KUKA KRL program: MyProgram_283().src

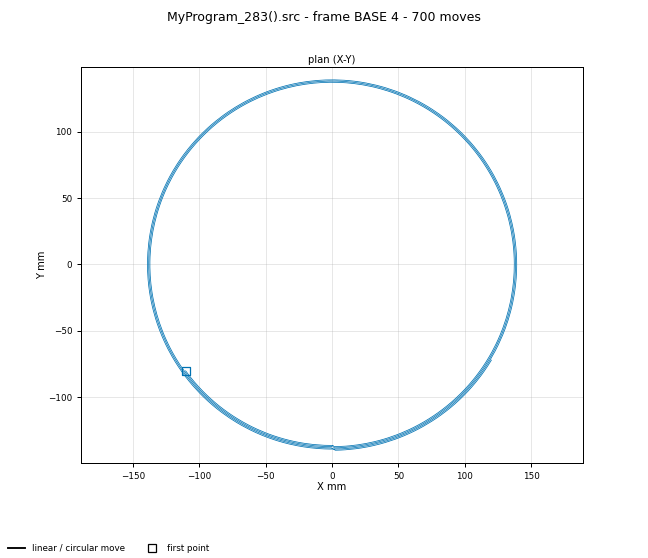
[picture p0: tool path of MyProgram_283().src in frame BASE 4, 700 of 700 moves have a stored position in this frame; points joined in program order, loops and branches not executed]
&ACCESS RVP
&REL 1
&PARAM TEMPLATE = C:\KRC\Roboter\Template\vorgabe
&PARAM EDITMASK = *
DEF MyProgram_283()
; ---- Setting reference (Base) ----
$BASE = BASE_DATA[4]

; --------------------------
; ---- Setting tool (TCP) ----
$TOOL = TOOL_DATA[3]
; --------------------------

$VEL.CP = VEL_APROX_PRINT
Startdeposition()
$VEL.CP = VEL_PRINT
LIN {X -110.2692,Y -80.0959,Z 174,A -140.9321,B 7.819,C 0.3265,E1 7.6978,E2 232.605} C_DIS
LIN {X -108.3483,Y -82.6759,Z 174,A -140.0536,B 7.8185,C 0.3365,E1 7.6992,E2 231.7869} C_DIS
LIN {X -106.4293,Y -85.1325,Z 174,A -138.4411,B 7.8186,C 0.3349,E1 7.7021,E2 230.1369} C_DIS
LIN {X -103.6871,Y -88.4515,Z 174,A -136.5544,B 7.8185,C 0.3377,E1 7.7055,E2 228.2411} C_DIS
LIN {X -100.4815,Y -92.0768,Z 174,A -134.4674,B 7.8184,C 0.3411,E1 7.7094,E2 226.1481} C_DIS
LIN {X -97.217,Y -95.517,Z 174,A -132.493,B 7.8182,C 0.3454,E1 7.7132,E2 224.1768} C_DIS
LIN {X -94.0859,Y -98.6027,Z 174,A -130.65,B 7.818,C 0.349,E1 7.7169,E2 222.335} C_DIS
LIN {X -91.5206,Y -100.9882,Z 174,A -129.1738,B 7.8179,C 0.3517,E1 7.7199,E2 220.8588} C_DIS
LIN {X -88.1965,Y -103.9039,Z 174,A -127.2223,B 7.8178,C 0.3537,E1 7.7241,E2 218.8959} C_DIS
LIN {X -85.404,Y -106.2113,Z 174,A -125.7546,B 7.8176,C 0.3571,E1 7.7273,E2 217.4355} C_DIS
LIN {X -81.9305,Y -108.9131,Z 174,A -123.8794,B 7.8176,C 0.3598,E1 7.7314,E2 215.5574} C_DIS
LIN {X -78.2052,Y -111.6189,Z 174,A -121.9045,B 7.8174,C 0.3623,E1 7.7359,E2 213.5778} C_DIS
LIN {X -74.5757,Y -114.0758,Z 174,A -119.9983,B 7.8174,C 0.3641,E1 7.7404,E2 211.6637} C_DIS
LIN {X -70.8017,Y -116.4554,Z 174,A -118.139,B 7.8172,C 0.367,E1 7.7448,E2 209.8066} C_DIS
LIN {X -67.0685,Y -118.6447,Z 174,A -116.2625,B 7.8172,C 0.3685,E1 7.7494,E2 207.9229} C_DIS
LIN {X -63.0831,Y -120.8085,Z 174,A -114.4681,B 7.8169,C 0.3727,E1 7.7537,E2 206.1427} C_DIS
LIN {X -59.9153,Y -122.4109,Z 174,A -112.95,B 7.8169,C 0.374,E1 7.7575,E2 204.6212} C_DIS
LIN {X -56.3626,Y -124.0885,Z 174,A -110.873,B 7.8171,C 0.369,E1 7.763,E2 202.4898} C_DIS
LIN {X -52.8036,Y -125.6422,Z 174,A -109.8689,B 7.8165,C 0.3809,E1 7.7653,E2 201.5659} C_DIS
LIN {X -50.2131,Y -126.7017,Z 174,A -108.4961,B 7.8166,C 0.3788,E1 7.769,E2 200.1681} C_DIS
LIN {X -47.4613,Y -127.7563,Z 174,A -107.243,B 7.8166,C 0.3797,E1 7.7722,E2 198.9129} C_DIS
LIN {X -43.8105,Y -129.0558,Z 174,A -105.3205,B 7.8167,C 0.3762,E1 7.7774,E2 196.9527} C_DIS
LIN {X -39.5544,Y -130.4212,Z 174,A -103.6952,B 7.8165,C 0.3818,E1 7.7817,E2 195.3594} C_DIS
LIN {X -36.2087,Y -131.39,Z 174,A -102.1521,B 7.8165,C 0.3815,E1 7.7858,E2 193.806} C_DIS
LIN {X -31.9644,Y -132.4856,Z 174,A -100.4334,B 7.8163,C 0.3847,E1 7.7905,E2 192.1027} C_DIS
LIN {X -28.5945,Y -133.2537,Z 174,A -98.9383,B 7.8163,C 0.3847,E1 7.7945,E2 190.6019} C_DIS
LIN {X -24.9403,Y -133.9873,Z 174,A -97.2215,B 7.8164,C 0.3828,E1 7.7993,E2 188.8655} C_DIS
LIN {X -20.6436,Y -134.7148,Z 174,A -95.52,B 7.8163,C 0.3857,E1 7.804,E2 187.18} C_DIS
LIN {X -13.919,Y -135.576,Z 174,A -92.555,B 7.8163,C 0.3844,E1 7.8122,E2 184.1995} C_DIS
LIN {X -5.8674,Y -136.1621,Z 174,A -88.2649,B 7.8171,C 0.3688,E1 7.8245,E2 179.7921} C_DIS
LIN {X 0.9737,Y -136.2785,Z 174,A -87.9401,B 7.8149,C 0.413,E1 7.8247,E2 179.7914} C_DIS
Enddeposition()
LIN {X 0.9737,Y -136.2785,Z 174,A -87.9404,B 7.8149,C 0.413,E1 7.8246,E2 179.7917} C_DIS
Startdeposition()
$VEL.CP = VEL_PRINT
LIN {X -0.4455,Y -137.1941,Z 174,A -87.6174,B 7.7989,C 0.4021,E1 7.8091,E2 179.393} C_DIS
LIN {X -3.8273,Y -137.1411,Z 174,A -88.9609,B 7.7989,C 0.401,E1 7.8053,E2 180.7283} C_DIS
LIN {X -6.8725,Y -137.0222,Z 174,A -90.2421,B 7.7989,C 0.4011,E1 7.8017,E2 182.0112} C_DIS
LIN {X -9.9728,Y -136.8314,Z 174,A -91.5485,B 7.7989,C 0.4011,E1 7.7981,E2 183.3192} C_DIS
LIN {X -13.3149,Y -136.5469,Z 174,A -93.0053,B 7.7989,C 0.4019,E1 7.794,E2 184.7837} C_DIS
LIN {X -17.0384,Y -136.1345,Z 174,A -94.5158,B 7.7989,C 0.4007,E1 7.7898,E2 186.288} C_DIS
LIN {X -19.6937,Y -135.7738,Z 174,A -95.6857,B 7.7989,C 0.4012,E1 7.7866,E2 187.4647} C_DIS
LIN {X -23.3734,Y -135.191,Z 174,A -97.2013,B 7.7989,C 0.4,E1 7.7824,E2 188.9758} C_DIS
LIN {X -25.9226,Y -134.723,Z 174,A -98.3187,B 7.7989,C 0.4001,E1 7.7793,E2 190.0978} C_DIS
LIN {X -29.7515,Y -133.9319,Z 174,A -99.9292,B 7.799,C 0.399,E1 7.775,E2 191.706} C_DIS
LIN {X -32.9498,Y -133.1812,Z 174,A -101.3082,B 7.799,C 0.3983,E1 7.7712,E2 193.0863} C_DIS
LIN {X -35.6372,Y -132.4851,Z 174,A -102.4768,B 7.799,C 0.3978,E1 7.768,E2 194.2562} C_DIS
LIN {X -39.3506,Y -131.4323,Z 174,A -104.0952,B 7.7991,C 0.3968,E1 7.7637,E2 195.8759} C_DIS
LIN {X -42.547,Y -130.4326,Z 174,A -105.5028,B 7.7991,C 0.3958,E1 7.76,E2 197.2848} C_DIS
LIN {X -45.2788,Y -129.5074,Z 174,A -106.7111,B 7.7992,C 0.3949,E1 7.7568,E2 198.4938} C_DIS
LIN {X -48.9163,Y -128.18,Z 174,A -108.344,B 7.7993,C 0.3937,E1 7.7525,E2 200.129} C_DIS
LIN {X -52.0827,Y -126.9264,Z 174,A -109.7771,B 7.7993,C 0.3925,E1 7.7488,E2 201.5636} C_DIS
LIN {X -55.2327,Y -125.5877,Z 174,A -111.2177,B 7.7994,C 0.3912,E1 7.7451,E2 203.0058} C_DIS
LIN {X -57.9714,Y -124.345,Z 174,A -112.4934,B 7.7994,C 0.3901,E1 7.7418,E2 204.284} C_DIS
LIN {X -61.4699,Y -122.6555,Z 174,A -114.1207,B 7.7996,C 0.3883,E1 7.7377,E2 205.912} C_DIS
LIN {X -64.5504,Y -121.0626,Z 174,A -115.5293,B 7.7996,C 0.3859,E1 7.7343,E2 207.3156} C_DIS
LIN {X -67.5416,Y -119.4194,Z 174,A -117.1085,B 7.7996,C 0.3865,E1 7.7304,E2 208.9142} C_DIS
LIN {X -71.3674,Y -117.1734,Z 174,A -118.9919,B 7.7998,C 0.3844,E1 7.7258,E2 210.8014} C_DIS
LIN {X -75.0753,Y -114.8329,Z 174,A -120.8424,B 7.7998,C 0.382,E1 7.7215,E2 212.6542} C_DIS
LIN {X -78.7185,Y -112.3668,Z 174,A -122.6965,B 7.8,C 0.3794,E1 7.7172,E2 214.5103} C_DIS
LIN {X -82.2906,Y -109.7778,Z 174,A -124.5598,B 7.8001,C 0.3768,E1 7.713,E2 216.3759} C_DIS
LIN {X -85.7856,Y -107.0689,Z 174,A -126.4313,B 7.8003,C 0.374,E1 7.7089,E2 218.2502} C_DIS
LIN {X -89.1974,Y -104.2437,Z 174,A -128.3004,B 7.8004,C 0.371,E1 7.7049,E2 220.1213} C_DIS
LIN {X -92.5203,Y -101.306,Z 174,A -130.1674,B 7.8006,C 0.3678,E1 7.701,E2 221.9898} C_DIS
LIN {X -95.7488,Y -98.2602,Z 174,A -132.0532,B 7.8007,C 0.3647,E1 7.6972,E2 223.8792} C_DIS
LIN {X -98.8778,Y -95.1109,Z 174,A -133.9317,B 7.8009,C 0.3614,E1 7.6936,E2 225.7601} C_DIS
LIN {X -101.9023,Y -91.8631,Z 174,A -135.8135,B 7.801,C 0.358,E1 7.69,E2 227.6449} C_DIS
LIN {X -104.8178,Y -88.5219,Z 174,A -137.691,B 7.8012,C 0.3545,E1 7.6866,E2 229.5249} C_DIS
LIN {X -107.6201,Y -85.093,Z 174,A -139.5665,B 7.8013,C 0.3508,E1 7.6833,E2 231.403} C_DIS
LIN {X -110.3053,Y -81.5822,Z 174,A -141.4389,B 7.8015,C 0.3471,E1 7.6801,E2 233.278} C_DIS
LIN {X -112.87,Y -77.9954,Z 174,A -143.3042,B 7.8017,C 0.3432,E1 7.6771,E2 235.1454} C_DIS
LIN {X -115.3112,Y -74.3387,Z 174,A -145.1385,B 7.8019,C 0.3388,E1 7.6743,E2 236.9785} C_DIS
LIN {X -117.6262,Y -70.6186,Z 174,A -147.0255,B 7.802,C 0.3352,E1 7.6716,E2 238.8718} C_DIS
LIN {X -119.8129,Y -66.8414,Z 174,A -148.8797,B 7.8022,C 0.3312,E1 7.669,E2 240.729} C_DIS
LIN {X -121.8696,Y -63.0137,Z 174,A -150.6229,B 7.8024,C 0.3256,E1 7.6668,E2 242.4622} C_DIS
LIN {X -123.252,Y -60.2605,Z 174,A -151.9559,B 7.8025,C 0.323,E1 7.6651,E2 243.8002} C_DIS
LIN {X -124.8864,Y -56.8005,Z 174,A -153.5542,B 7.8027,C 0.3189,E1 7.6632,E2 245.3976} C_DIS
LIN {X -126.2078,Y -53.7984,Z 174,A -154.9308,B 7.8028,C 0.3154,E1 7.6617,E2 246.7743} C_DIS
LIN {X -127.5638,Y -50.5013,Z 174,A -156.4598,B 7.803,C 0.3121,E1 7.6601,E2 248.3074} C_DIS
LIN {X -128.7749,Y -47.3279,Z 174,A -157.9017,B 7.8031,C 0.3086,E1 7.6587,E2 249.7512} C_DIS
LIN {X -129.8649,Y -44.2476,Z 174,A -159.2776,B 7.8032,C 0.3051,E1 7.6574,E2 251.1276} C_DIS
LIN {X -130.9429,Y -40.9494,Z 174,A -160.7629,B 7.8034,C 0.3016,E1 7.6561,E2 252.6164} C_DIS
LIN {X -131.9007,Y -37.7508,Z 174,A -162.1808,B 7.8035,C 0.2981,E1 7.655,E2 254.0363} C_DIS
LIN {X -132.775,Y -34.55,Z 174,A -163.5899,B 7.8036,C 0.2946,E1 7.654,E2 255.4473} C_DIS
LIN {X -133.5558,Y -31.3956,Z 174,A -164.9673,B 7.8038,C 0.2911,E1 7.6531,E2 256.8263} C_DIS
LIN {X -134.2131,Y -28.4489,Z 174,A -166.2332,B 7.8039,C 0.2877,E1 7.6524,E2 258.0917} C_DIS
LIN {X -134.9062,Y -24.9647,Z 174,A -167.9218,B 7.8039,C 0.2863,E1 7.6515,E2 259.8047} C_DIS
LIN {X -135.5635,Y -21.0908,Z 174,A -169.4474,B 7.8042,C 0.2801,E1 7.6508,E2 261.3146} C_DIS
LIN {X -136.0332,Y -17.8113,Z 174,A -170.838,B 7.8043,C 0.2762,E1 7.6502,E2 262.705} C_DIS
LIN {X -136.4086,Y -14.6623,Z 174,A -172.1793,B 7.8044,C 0.2727,E1 7.6498,E2 264.0473} C_DIS
LIN {X -136.7046,Y -11.5825,Z 174,A -173.5097,B 7.8045,C 0.2695,E1 7.6495,E2 265.3814} C_DIS
LIN {X -136.9358,Y -8.4199,Z 174,A -174.8471,B 7.8047,C 0.2659,E1 7.6492,E2 266.7192} C_DIS
LIN {X -137.0908,Y -5.331,Z 174,A -176.155,B 7.8047,C 0.2624,E1 7.6491,E2 268.0281} C_DIS
LIN {X -137.1758,Y -2.2664,Z 174,A -177.5113,B 7.8049,C 0.2598,E1 7.649,E2 269.3927} C_DIS
LIN {X -137.1758,Y 2.2664,Z 174,A -179.4228,B 7.805,C 0.2546,E1 7.649,E2 271.3049} C_DIS
LIN {X -137.0733,Y 5.7817,Z 174,A 179.0821,B 7.8052,C 0.2507,E1 7.6492,E2 272.8019} C_DIS
LIN {X -136.8871,Y 9.2111,Z 174,A 177.6403,B 7.8052,C 0.2467,E1 7.6494,E2 274.2435} C_DIS
LIN {X -136.6416,Y 12.3277,Z 174,A 176.3073,B 7.8054,C 0.2433,E1 7.6497,E2 275.5787} C_DIS
LIN {X -136.3398,Y 15.3018,Z 174,A 175.0369,B 7.8055,C 0.24,E1 7.6501,E2 276.8506} C_DIS
LIN {X -135.9783,Y 18.2303,Z 174,A 173.7751,B 7.8055,C 0.2369,E1 7.6505,E2 278.1149} C_DIS
LIN {X -135.456,Y 21.7848,Z 174,A 172.2427,B 7.8057,C 0.233,E1 7.6512,E2 279.6498} C_DIS
LIN {X -134.9062,Y 24.9647,Z 174,A 170.8671,B 7.8058,C 0.2296,E1 7.6519,E2 281.0276} C_DIS
LIN {X -134.2768,Y 28.1541,Z 174,A 169.4815,B 7.8059,C 0.2261,E1 7.6526,E2 282.4155} C_DIS
LIN {X -133.5668,Y 31.3501,Z 174,A 168.0864,B 7.806,C 0.2227,E1 7.6535,E2 283.8127} C_DIS
LIN {X -132.775,Y 34.55,Z 174,A 166.6818,B 7.8061,C 0.2192,E1 7.6545,E2 285.2193} C_DIS
LIN {X -131.9007,Y 37.7508,Z 174,A 165.2679,B 7.8062,C 0.2157,E1 7.6555,E2 286.6354} C_DIS
LIN {X -131.118,Y 40.3774,Z 174,A 164.0773,B 7.8062,C 0.2131,E1 7.6565,E2 287.8305} C_DIS
LIN {X -129.9012,Y 44.1428,Z 174,A 162.4156,B 7.8064,C 0.2087,E1 7.658,E2 289.4918} C_DIS
LIN {X -128.7749,Y 47.3279,Z 174,A 160.977,B 7.8064,C 0.2053,E1 7.6593,E2 290.9324} C_DIS
LIN {X -127.5638,Y 50.5013,Z 174,A 159.5313,B 7.8066,C 0.2018,E1 7.6608,E2 292.3801} C_DIS
LIN {X -126.2676,Y 53.66,Z 174,A 158.0783,B 7.8066,C 0.1984,E1 7.6624,E2 293.835} C_DIS
LIN {X -124.8864,Y 56.8005,Z 174,A 156.6188,B 7.8068,C 0.195,E1 7.664,E2 295.2964} C_DIS
LIN {X -123.4203,Y 59.9195,Z 174,A 155.1528,B 7.8068,C 0.1916,E1 7.6658,E2 296.7643} C_DIS
LIN {X -121.8696,Y 63.0137,Z 174,A 153.6811,B 7.8069,C 0.1882,E1 7.6677,E2 298.2377} C_DIS
LIN {X -120.4387,Y 65.7058,Z 174,A 152.3208,B 7.8069,C 0.1862,E1 7.6695,E2 299.6074} C_DIS
LIN {X -118.2905,Y 69.4987,Z 174,A 150.4681,B 7.8071,C 0.182,E1 7.6721,E2 301.4623} C_DIS
LIN {X -116.0135,Y 73.2364,Z 174,A 148.6087,B 7.8071,C 0.178,E1 7.6748,E2 303.3238} C_DIS
LIN {X -113.6097,Y 76.9126,Z 174,A 146.7435,B 7.8072,C 0.174,E1 7.6777,E2 305.191} C_DIS
LIN {X -111.1522,Y 80.4234,Z 174,A 144.8998,B 7.8073,C 0.1705,E1 7.6807,E2 307.0395} C_DIS
LIN {X -108.4431,Y 84.0405,Z 174,A 143.0035,B 7.8074,C 0.1663,E1 7.6839,E2 308.9351} C_DIS
LIN {X -105.6641,Y 87.5089,Z 174,A 141.1225,B 7.8074,C 0.1624,E1 7.6872,E2 310.8174} C_DIS
LIN {X -102.7942,Y 90.8629,Z 174,A 139.2504,B 7.8076,C 0.1588,E1 7.6906,E2 312.6912} C_DIS
LIN {X -99.7895,Y 94.1529,Z 174,A 137.3641,B 7.8076,C 0.1552,E1 7.6942,E2 314.5788} C_DIS
LIN {X -96.7042,Y 97.3191,Z 174,A 135.4889,B 7.8077,C 0.1518,E1 7.6979,E2 316.4558} C_DIS
LIN {X -93.5053,Y 100.3966,Z 174,A 133.6105,B 7.8077,C 0.1485,E1 7.7017,E2 318.3355} C_DIS
LIN {X -90.1964,Y 103.3795,Z 174,A 131.7333,B 7.8078,C 0.1451,E1 7.7056,E2 320.213} C_DIS
LIN {X -86.8106,Y 106.2386,Z 174,A 129.8571,B 7.8078,C 0.1421,E1 7.7097,E2 322.0907} C_DIS
LIN {X -83.3398,Y 108.9825,Z 174,A 127.9883,B 7.8079,C 0.1391,E1 7.7138,E2 323.9604} C_DIS
LIN {X -79.7901,Y 111.6076,Z 174,A 126.1244,B 7.8079,C 0.1362,E1 7.718,E2 325.8252} C_DIS
LIN {X -76.1826,Y 114.1005,Z 174,A 124.2709,B 7.808,C 0.1336,E1 7.7223,E2 327.6797} C_DIS
LIN {X -72.4936,Y 116.4792,Z 174,A 122.4202,B 7.808,C 0.131,E1 7.7266,E2 329.531} C_DIS
LIN {X -68.7443,Y 118.7305,Z 174,A 120.5776,B 7.8081,C 0.1285,E1 7.7311,E2 331.3741} C_DIS
LIN {X -65.1753,Y 120.7269,Z 174,A 118.7981,B 7.8081,C 0.1272,E1 7.7354,E2 333.1609} C_DIS
LIN {X -61.6024,Y 122.588,Z 174,A 117.2225,B 7.8082,C 0.1234,E1 7.7393,E2 334.7222} C_DIS
LIN {X -58.3628,Y 124.164,Z 174,A 115.7112,B 7.8082,C 0.1216,E1 7.7431,E2 336.2332} C_DIS
LIN {X -55.5354,Y 125.4523,Z 174,A 114.3848,B 7.8082,C 0.1205,E1 7.7465,E2 337.562} C_DIS
LIN {X -52.0827,Y 126.9264,Z 174,A 112.8269,B 7.8082,C 0.1186,E1 7.7505,E2 339.1176} C_DIS
LIN {X -49.2458,Y 128.0519,Z 174,A 111.5224,B 7.8082,C 0.1177,E1 7.7539,E2 340.4247} C_DIS
LIN {X -45.7366,Y 129.3487,Z 174,A 109.9741,B 7.8083,C 0.1159,E1 7.758,E2 341.9702} C_DIS
LIN {X -43.1013,Y 130.248,Z 174,A 108.7904,B 7.8083,C 0.1152,E1 7.7611,E2 343.1556} C_DIS
LIN {X -39.7978,Y 131.2954,Z 174,A 107.3456,B 7.8083,C 0.1139,E1 7.765,E2 344.5991} C_DIS
LIN {X -36.1505,Y 132.3482,Z 174,A 105.7605,B 7.8083,C 0.1126,E1 7.7692,E2 346.1832} C_DIS
LIN {X -33.2373,Y 133.1082,Z 174,A 104.5097,B 7.8083,C 0.1116,E1 7.7726,E2 347.4323} C_DIS
LIN {X -29.7515,Y 133.9319,Z 174,A 102.9992,B 7.8083,C 0.1109,E1 7.7767,E2 348.9437} C_DIS
LIN {X -26.5584,Y 134.6015,Z 174,A 101.6336,B 7.8083,C 0.1102,E1 7.7805,E2 350.3089} C_DIS
LIN {X -23.3734,Y 135.191,Z 174,A 100.2786,B 7.8084,C 0.1095,E1 7.7842,E2 351.6634} C_DIS
LIN {X -20.5736,Y 135.6436,Z 174,A 99.1141,B 7.8084,C 0.1086,E1 7.7874,E2 352.8246} C_DIS
LIN {X -17.0384,Y 136.1345,Z 174,A 97.601,B 7.8084,C 0.1084,E1 7.7916,E2 354.3398} C_DIS
LIN {X -13.8935,Y 136.4913,Z 174,A 96.2787,B 7.8084,C 0.108,E1 7.7952,E2 355.6614} C_DIS
LIN {X -10.7669,Y 136.7735,Z 174,A 94.9682,B 7.8084,C 0.1077,E1 7.7989,E2 356.9712} C_DIS
LIN {X -7.6609,Y 136.9826,Z 174,A 93.6688,B 7.8084,C 0.1074,E1 7.8025,E2 358.2698} C_DIS
LIN {X -4.6128,Y 137.1189,Z 174,A 92.3958,B 7.8084,C 0.1073,E1 7.8061,E2 359.542} C_DIS
LIN {X -1.5193,Y 137.1882,Z 174,A 91.1061,B 7.8084,C 0.1072,E1 7.8097,E2 360.8308} C_DIS
LIN {X 1.5193,Y 137.1882,Z 174,A 89.8358,B 7.8084,C 0.1072,E1 7.8132,E2 362.1007} C_DIS
LIN {X 4.5776,Y 137.1202,Z 174,A 88.5564,B 7.8084,C 0.1073,E1 7.8168,E2 363.3799} C_DIS
LIN {X 7.6609,Y 136.9826,Z 174,A 87.2662,B 7.8084,C 0.1075,E1 7.8204,E2 364.6696} C_DIS
LIN {X 10.7669,Y 136.7735,Z 174,A 85.9654,B 7.8084,C 0.1078,E1 7.824,E2 365.9701} C_DIS
LIN {X 13.8935,Y 136.4913,Z 174,A 84.6542,B 7.8084,C 0.1082,E1 7.8276,E2 367.2808} C_DIS
LIN {X 16.4844,Y 136.2006,Z 174,A 83.5114,B 7.8084,C 0.1094,E1 7.8308,E2 368.4298} C_DIS
LIN {X 20.1992,Y 135.7015,Z 174,A 82.0017,B 7.8084,C 0.1091,E1 7.835,E2 369.9322} C_DIS
LIN {X 23.02,Y 135.2499,Z 174,A 80.8055,B 7.8084,C 0.1097,E1 7.8383,E2 371.1284} C_DIS
LIN {X 26.5584,Y 134.6015,Z 174,A 79.3107,B 7.8084,C 0.1104,E1 7.8424,E2 372.6219} C_DIS
LIN {X 29.7515,Y 133.9319,Z 174,A 77.9513,B 7.8084,C 0.1112,E1 7.8461,E2 373.9806} C_DIS
LIN {X 32.4849,Y 133.2932,Z 174,A 76.7795,B 7.8084,C 0.1119,E1 7.8493,E2 375.1519} C_DIS
LIN {X 36.1505,Y 132.3482,Z 174,A 75.2069,B 7.8084,C 0.1129,E1 7.8535,E2 376.7233} C_DIS
LIN {X 39.3506,Y 131.4323,Z 174,A 73.8223,B 7.8084,C 0.114,E1 7.8572,E2 378.107} C_DIS
LIN {X 42.1496,Y 130.5595,Z 174,A 72.6051,B 7.8084,C 0.1149,E1 7.8605,E2 379.323} C_DIS
LIN {X 45.3005,Y 129.4999,Z 174,A 71.184,B 7.8084,C 0.1168,E1 7.8642,E2 380.7478} C_DIS
LIN {X 48.9163,Y 128.18,Z 174,A 69.6223,B 7.8083,C 0.1176,E1 7.8683,E2 382.3038} C_DIS
LIN {X 52.0827,Y 126.9264,Z 174,A 68.2082,B 7.8083,C 0.1189,E1 7.872,E2 383.7168} C_DIS
LIN {X 54.7796,Y 125.7835,Z 174,A 66.971,B 7.8083,C 0.1206,E1 7.8751,E2 384.9555} C_DIS
LIN {X 58.3628,Y 124.164,Z 174,A 65.3616,B 7.8083,C 0.1219,E1 7.8792,E2 386.561} C_DIS
LIN {X 61.4699,Y 122.6555,Z 174,A 63.9296,B 7.8082,C 0.1236,E1 7.8828,E2 387.9916} C_DIS
LIN {X 65.316,Y 120.6513,Z 174,A 62.0347,B 7.8082,C 0.1275,E1 7.8875,E2 389.8968} C_DIS
LIN {X 69.1142,Y 118.5164,Z 174,A 60.2332,B 7.8081,C 0.1298,E1 7.8919,E2 391.6961} C_DIS
LIN {X 72.8152,Y 116.279,Z 174,A 58.4343,B 7.8081,C 0.1324,E1 7.8961,E2 393.4943} C_DIS
LIN {X 76.5407,Y 113.8614,Z 174,A 56.6028,B 7.8081,C 0.1349,E1 7.9004,E2 395.3232} C_DIS
LIN {X 80.1165,Y 111.3742,Z 174,A 54.8001,B 7.808,C 0.1376,E1 7.9045,E2 397.1241} C_DIS
LIN {X 83.6439,Y 108.75,Z 174,A 52.981,B 7.808,C 0.1404,E1 7.9086,E2 398.9413} C_DIS
LIN {X 87.1606,Y 105.9525,Z 174,A 51.1526,B 7.8079,C 0.1429,E1 7.9125,E2 400.7642} C_DIS
LIN {X 90.5375,Y 103.0819,Z 174,A 49.3008,B 7.8079,C 0.1464,E1 7.9164,E2 402.6166} C_DIS
LIN {X 93.8233,Y 100.1004,Z 174,A 47.474,B 7.8077,C 0.1495,E1 7.9202,E2 404.4406} C_DIS
LIN {X 97.0127,Y 97.0127,Z 174,A 45.6408,B 7.8077,C 0.1528,E1 7.9238,E2 406.2718} C_DIS
LIN {X 100.1004,Y 93.8233,Z 174,A 43.8151,B 7.8077,C 0.1561,E1 7.9273,E2 408.0947} C_DIS
LIN {X 103.0484,Y 90.5753,Z 174,A 42.0001,B 7.8075,C 0.1597,E1 7.9307,E2 409.9081} C_DIS
LIN {X 105.9525,Y 87.1606,Z 174,A 40.1605,B 7.8075,C 0.1632,E1 7.934,E2 411.7444} C_DIS
LIN {X 108.7084,Y 83.6982,Z 174,A 38.3433,B 7.8075,C 0.1668,E1 7.9371,E2 413.5585} C_DIS
LIN {X 111.3458,Y 80.1562,Z 174,A 36.5276,B 7.8073,C 0.1705,E1 7.9401,E2 415.3716} C_DIS
LIN {X 113.8614,Y 76.5407,Z 174,A 34.7284,B 7.8073,C 0.174,E1 7.9429,E2 417.1667} C_DIS
LIN {X 116.2257,Y 72.9003,Z 174,A 32.9254,B 7.8071,C 0.1782,E1 7.9456,E2 418.9693} C_DIS
LIN {X 118.5164,Y 69.1142,Z 174,A 31.1171,B 7.8071,C 0.182,E1 7.9482,E2 420.7737} C_DIS
LIN {X 120.6905,Y 65.243,Z 174,A 29.2721,B 7.807,C 0.1865,E1 7.9507,E2 422.6184} C_DIS
LIN {X 122.6555,Y 61.4699,Z 174,A 27.6419,B 7.807,C 0.1881,E1 7.9528,E2 424.2315} C_DIS
LIN {X 124.06,Y 58.5804,Z 174,A 26.3164,B 7.8068,C 0.1913,E1 7.9544,E2 425.5558} C_DIS
LIN {X 125.5877,Y 55.2327,Z 174,A 24.8144,B 7.8068,C 0.1946,E1 7.9561,E2 427.0544} C_DIS
LIN {X 126.9264,Y 52.0827,Z 174,A 23.4107,B 7.8067,C 0.1979,E1 7.9576,E2 428.4558} C_DIS
LIN {X 128.18,Y 48.9163,Z 174,A 22.0147,B 7.8066,C 0.2012,E1 7.959,E2 429.8495} C_DIS
LIN {X 129.3071,Y 45.852,Z 174,A 20.6839,B 7.8066,C 0.2042,E1 7.9602,E2 431.177} C_DIS
LIN {X 130.291,Y 42.9722,Z 174,A 19.3951,B 7.8064,C 0.208,E1 7.9614,E2 432.4689} C_DIS
LIN {X 131.4323,Y 39.3506,Z 174,A 17.8735,B 7.8064,C 0.2111,E1 7.9626,E2 433.9837} C_DIS
LIN {X 132.2311,Y 36.5694,Z 174,A 16.7076,B 7.8063,C 0.2136,E1 7.9635,E2 435.145} C_DIS
LIN {X 133.0818,Y 33.3411,Z 174,A 15.2919,B 7.8061,C 0.2179,E1 7.9645,E2 436.5644} C_DIS
LIN {X 133.9319,Y 29.7515,Z 174,A 13.81,B 7.8061,C 0.221,E1 7.9654,E2 438.0403} C_DIS
LIN {X 134.5149,Y 26.9838,Z 174,A 12.6419,B 7.806,C 0.2241,E1 7.9661,E2 439.2076} C_DIS
LIN {X 135.1366,Y 23.6773,Z 174,A 11.2568,B 7.8059,C 0.2277,E1 7.9668,E2 440.5912} C_DIS
LIN {X 135.7015,Y 20.1992,Z 174,A 9.8324,B 7.8058,C 0.2309,E1 7.9674,E2 442.011} C_DIS
LIN {X 136.1345,Y 17.0384,Z 174,A 8.5267,B 7.8057,C 0.2342,E1 7.9679,E2 443.3145} C_DIS
LIN {X 136.4913,Y 13.8935,Z 174,A 7.2313,B 7.8056,C 0.2374,E1 7.9683,E2 444.6076} C_DIS
LIN {X 136.7233,Y 11.3606,Z 174,A 6.1315,B 7.8055,C 0.2412,E1 7.9685,E2 445.713} C_DIS
LIN {X 136.9826,Y 7.6609,Z 174,A 4.6731,B 7.8054,C 0.2439,E1 7.9688,E2 447.1614} C_DIS
LIN {X 137.1352,Y 4.0399,Z 174,A 3.1415,B 7.8052,C 0.2486,E1 7.9689,E2 448.6964} C_DIS
LIN {X 137.196,Y 0.3997,Z 174,A 1.6281,B 7.8052,C 0.2528,E1 7.9689,E2 450.2104} C_DIS
LIN {X 137.1628,Y -3.0452,Z 174,A 0.2856,B 7.805,C 0.2551,E1 7.9689,E2 451.5421} C_DIS
LIN {X 137.0602,Y -6.1163,Z 174,A -0.9764,B 7.805,C 0.2583,E1 7.9688,E2 452.8026} C_DIS
LIN {X 136.8871,Y -9.2111,Z 174,A -2.2496,B 7.8048,C 0.2616,E1 7.9686,E2 454.0743} C_DIS
LIN {X 136.6416,Y -12.3277,Z 174,A -3.5333,B 7.8048,C 0.2649,E1 7.9683,E2 455.3563} C_DIS
LIN {X 136.3336,Y -15.3591,Z 174,A -4.7733,B 7.8046,C 0.268,E1 7.9679,E2 456.5935} C_DIS
LIN {X 135.9276,Y -18.6169,Z 174,A -6.133,B 7.8045,C 0.2717,E1 7.9674,E2 457.9529} C_DIS
LIN {X 135.456,Y -21.7848,Z 174,A -7.448,B 7.8044,C 0.275,E1 7.9668,E2 459.2664} C_DIS
LIN {X 134.9062,Y -24.9647,Z 174,A -8.7732,B 7.8042,C 0.2784,E1 7.9662,E2 460.59} C_DIS
LIN {X 134.3758,Y -27.6674,Z 174,A -9.9471,B 7.8042,C 0.2822,E1 7.9655,E2 461.7679} C_DIS
LIN {X 133.5668,Y -31.3501,Z 174,A -11.4528,B 7.804,C 0.2852,E1 7.9646,E2 463.2664} C_DIS
LIN {X 132.8048,Y -34.4326,Z 174,A -12.7599,B 7.8039,C 0.2886,E1 7.9637,E2 464.5725} C_DIS
LIN {X 131.9007,Y -37.7508,Z 174,A -14.1696,B 7.8037,C 0.2921,E1 7.9627,E2 465.9802} C_DIS
LIN {X 130.9429,Y -40.9494,Z 174,A -15.541,B 7.8037,C 0.2955,E1 7.9616,E2 467.35} C_DIS
LIN {X 129.9012,Y -44.1428,Z 174,A -16.9205,B 7.8035,C 0.2989,E1 7.9603,E2 468.7279} C_DIS
LIN {X 128.7749,Y -47.3279,Z 174,A -18.3084,B 7.8034,C 0.3023,E1 7.959,E2 470.1144} C_DIS
LIN {X 127.6321,Y -50.3256,Z 174,A -19.6165,B 7.8032,C 0.3053,E1 7.9577,E2 471.4198} C_DIS
LIN {X 126.2676,Y -53.66,Z 174,A -21.1065,B 7.8031,C 0.3091,E1 7.9561,E2 472.9094} C_DIS
LIN {X 124.8864,Y -56.8005,Z 174,A -22.5161,B 7.803,C 0.3124,E1 7.9545,E2 474.3175} C_DIS
LIN {X 123.4203,Y -59.9195,Z 174,A -23.9324,B 7.8028,C 0.3158,E1 7.9528,E2 475.7324} C_DIS
LIN {X 121.8696,Y -63.0137,Z 174,A -25.3549,B 7.8027,C 0.3191,E1 7.951,E2 477.1533} C_DIS
LIN {X 120.4387,Y -65.7058,Z 174,A -26.6698,B 7.8025,C 0.3232,E1 7.9493,E2 478.4748} C_DIS
LIN {X 118.2905,Y -69.4987,Z 174,A -28.4621,B 7.8024,C 0.3273,E1 7.9468,E2 480.2653} C_DIS
LIN {X 116.0135,Y -73.2364,Z 174,A -30.262,B 7.8022,C 0.3313,E1 7.9441,E2 482.0635} C_DIS
LIN {X 113.6097,Y -76.9126,Z 174,A -32.0686,B 7.802,C 0.3353,E1 7.9413,E2 483.8684} C_DIS
LIN {X 111.0923,Y -80.506,Z 174,A -33.8771,B 7.8018,C 0.3392,E1 7.9384,E2 485.6757} C_DIS
LIN {X 108.4431,Y -84.0405,Z 174,A -35.6948,B 7.8017,C 0.343,E1 7.9353,E2 487.4918} C_DIS
LIN {X 105.6641,Y -87.5089,Z 174,A -37.5207,B 7.8015,C 0.3467,E1 7.9321,E2 489.3156} C_DIS
LIN {X 102.7942,Y -90.8629,Z 174,A -39.3416,B 7.8014,C 0.3504,E1 7.9288,E2 491.1354} C_DIS
LIN {X 99.7895,Y -94.1529,Z 174,A -41.1729,B 7.8012,C 0.3539,E1 7.9253,E2 492.9648} C_DIS
LIN {X 96.7515,Y -97.2722,Z 174,A -42.983,B 7.801,C 0.3576,E1 7.9218,E2 494.7756} C_DIS
LIN {X 93.5053,Y -100.3966,Z 174,A -44.8265,B 7.8009,C 0.3607,E1 7.918,E2 496.616} C_DIS
LIN {X 90.1964,Y -103.3795,Z 174,A -46.6592,B 7.8007,C 0.3639,E1 7.9142,E2 498.4469} C_DIS
LIN {X 86.911,Y -106.1565,Z 174,A -48.4587,B 7.8006,C 0.3674,E1 7.9103,E2 500.2484} C_DIS
LIN {X 83.3398,Y -108.9825,Z 174,A -50.3112,B 7.8005,C 0.37,E1 7.9063,E2 502.0964} C_DIS
LIN {X 79.7901,Y -111.6076,Z 174,A -52.133,B 7.8003,C 0.3729,E1 7.9021,E2 503.917} C_DIS
LIN {X 76.2021,Y -114.0875,Z 174,A -53.9411,B 7.8002,C 0.3757,E1 7.898,E2 505.7251} C_DIS
LIN {X 72.4936,Y -116.4792,Z 174,A -55.7587,B 7.8001,C 0.3783,E1 7.8937,E2 507.541} C_DIS
LIN {X 68.7443,Y -118.7305,Z 174,A -57.565,B 7.7999,C 0.3807,E1 7.8893,E2 509.3463} C_DIS
LIN {X 64.9253,Y -120.8612,Z 174,A -59.3579,B 7.7999,C 0.3828,E1 7.885,E2 511.1365} C_DIS
LIN {X 61.4699,Y -122.6555,Z 174,A -60.9165,B 7.7998,C 0.3839,E1 7.8811,E2 512.6879} C_DIS
LIN {X 58.3628,Y -124.164,Z 174,A -62.3451,B 7.7998,C 0.3856,E1 7.8775,E2 514.1158} C_DIS
LIN {X 55.2327,Y -125.5877,Z 174,A -63.7677,B 7.7996,C 0.3871,E1 7.8739,E2 515.5378} C_DIS
LIN {X 52.4956,Y -126.7539,Z 174,A -65.033,B 7.7996,C 0.3891,E1 7.8706,E2 516.8069} C_DIS
LIN {X 48.9163,Y -128.18,Z 174,A -66.5941,B 7.7995,C 0.3901,E1 7.8666,E2 518.3632} C_DIS
LIN {X 45.7366,Y -129.3487,Z 174,A -67.9974,B 7.7995,C 0.3914,E1 7.8629,E2 519.7661} C_DIS
LIN {X 42.547,Y -130.4326,Z 174,A -69.3929,B 7.7994,C 0.3926,E1 7.8592,E2 521.1612} C_DIS
LIN {X 39.5764,Y -131.3631,Z 174,A -70.6937,B 7.7993,C 0.3939,E1 7.8557,E2 522.4629} C_DIS
LIN {X 36.1505,Y -132.3482,Z 174,A -72.1614,B 7.7993,C 0.3948,E1 7.8518,E2 523.929} C_DIS
LIN {X 32.1666,Y -133.37,Z 174,A -73.8669,B 7.7992,C 0.396,E1 7.8471,E2 525.634} C_DIS
LIN {X 28.9694,Y -134.1008,Z 174,A -75.2342,B 7.7992,C 0.397,E1 7.8434,E2 527.0019} C_DIS
LIN {X 25.7781,Y -134.7507,Z 174,A -76.5797,B 7.7992,C 0.3976,E1 7.8397,E2 528.3465} C_DIS
LIN {X 22.5956,Y -135.3207,Z 174,A -77.9225,B 7.7991,C 0.3983,E1 7.836,E2 529.6891} C_DIS
LIN {X 19.4245,Y -135.8122,Z 174,A -79.2619,B 7.7991,C 0.399,E1 7.8323,E2 531.0292} C_DIS
LIN {X 16.2347,Y -136.2304,Z 174,A -80.5926,B 7.7991,C 0.3995,E1 7.8287,E2 532.359} C_DIS
LIN {X 13.1269,Y -136.5649,Z 174,A -81.8919,B 7.799,C 0.3999,E1 7.825,E2 533.6583} C_DIS
LIN {X 9.9728,Y -136.8314,Z 174,A -83.2417,B 7.799,C 0.4008,E1 7.8213,E2 535.0124} C_DIS
LIN {X 6.1163,Y -137.0602,Z 174,A -84.8167,B 7.799,C 0.4006,E1 7.8169,E2 536.5834} C_DIS
LIN {X 3.0452,Y -137.1628,Z 174,A -86.0956,B 7.799,C 0.4008,E1 7.8133,E2 537.8624} C_DIS
LIN {X 0.9766,Y -137.1895,Z 174,A -86.8725,B 7.799,C 0.3994,E1 7.8112,E2 538.6284} C_DIS
Enddeposition()
LIN {X 0.9766,Y -137.1895,Z 174,A -86.8725,B 7.799,C 0.3994,E1 7.8112,E2 538.6284} C_DIS
Startdeposition()
$VEL.CP = VEL_PRINT
LIN {X 1.6084,Y -138.094,Z 174,A -85.9601,B 7.782,C 0.3926,E1 7.7965,E2 537.6704} C_DIS
LIN {X 5.5097,Y -137.9917,Z 174,A -84.4095,B 7.782,C 0.3935,E1 7.8008,E2 536.1279} C_DIS
LIN {X 9.8394,Y -137.7507,Z 174,A -82.6213,B 7.782,C 0.3931,E1 7.8058,E2 534.3401} C_DIS
LIN {X 13.4506,Y -137.4451,Z 174,A -81.1698,B 7.782,C 0.3935,E1 7.8098,E2 532.8947} C_DIS
LIN {X 16.6463,Y -137.0948,Z 174,A -79.0849,B 7.7826,C 0.3792,E1 7.8159,E2 530.7105} C_DIS
LIN {X 22.351,Y -136.2812,Z 174,A -77.6149,B 7.7818,C 0.3947,E1 7.8196,E2 529.3597} C_DIS
LIN {X 26.3325,Y -135.5682,Z 174,A -75.8066,B 7.782,C 0.3912,E1 7.8246,E2 527.5335} C_DIS
LIN {X 29.4156,Y -134.9325,Z 174,A -74.4572,B 7.7821,C 0.3895,E1 7.8283,E2 526.1776} C_DIS
LIN {X 34.0037,Y -133.8496,Z 174,A -72.5109,B 7.7821,C 0.3881,E1 7.8336,E2 524.2312} C_DIS
LIN {X 37.0264,Y -133.0452,Z 174,A -71.2168,B 7.7822,C 0.3871,E1 7.8371,E2 522.9367} C_DIS
LIN {X 40.3618,Y -132.0714,Z 174,A -69.8055,B 7.7822,C 0.3863,E1 7.8408,E2 521.5284} C_DIS
LIN {X 45.7189,Y -130.3149,Z 174,A -67.4739,B 7.7824,C 0.384,E1 7.847,E2 519.1961} C_DIS
LIN {X 50.7038,Y -128.4581,Z 174,A -65.3045,B 7.7824,C 0.3822,E1 7.8527,E2 517.03} C_DIS
LIN {X 53.4133,Y -127.3537,Z 174,A -63.8756,B 7.7827,C 0.3767,E1 7.8564,E2 515.572} C_DIS
LIN {X 58.3037,Y -125.1907,Z 174,A -61.8635,B 7.7827,C 0.3777,E1 7.8615,E2 513.5852} C_DIS
LIN {X 61.9206,Y -123.4439,Z 174,A -60.2432,B 7.7827,C 0.3763,E1 7.8655,E2 511.9696} C_DIS
LIN {X 65.5374,Y -121.5621,Z 174,A -58.4935,B 7.7829,C 0.3728,E1 7.8699,E2 510.2109} C_DIS
LIN {X 69.2755,Y -119.4712,Z 174,A -56.4123,B 7.7833,C 0.3642,E1 7.875,E2 508.0884} C_DIS
LIN {X 72.5939,Y -117.4851,Z 174,A -55.0773,B 7.7833,C 0.3668,E1 7.8781,E2 506.7872} C_DIS
LIN {X 76.3802,Y -115.0593,Z 174,A -53.2717,B 7.7833,C 0.3649,E1 7.8823,E2 504.9878} C_DIS
LIN {X 80.6698,Y -112.0938,Z 174,A -50.14,B 7.7843,C 0.342,E1 7.8897,E2 501.727} C_DIS
LIN {X 86.7659,Y -107.4436,Z 174,A -48.4205,B 7.7833,C 0.3649,E1 7.8931,E2 500.1961} C_DIS
LIN {X 92.5399,Y -102.5131,Z 174,A -45.1507,B 7.7837,C 0.3564,E1 7.9001,E2 496.9081} C_DIS
LIN {X 96.8835,Y -98.4179,Z 174,A -42.5618,B 7.784,C 0.3491,E1 7.9053,E2 494.3024} C_DIS
LIN {X 102.454,Y -92.6051,Z 174,A -38.932,B 7.7846,C 0.3361,E1 7.9123,E2 490.6319} C_DIS
LIN {X 104.6651,Y -90.0981,Z 174,A -37.8424,B 7.7845,C 0.3389,E1 7.9143,E2 489.5797} C_DIS
LIN {X 107.2864,Y -86.9608,Z 174,A -35.7737,B 7.7849,C 0.3275,E1 7.918,E2 487.4609} C_DIS
LIN {X 109.7627,Y -83.813,Z 174,A -34.62,B 7.7847,C 0.3339,E1 7.9199,E2 486.3716} C_DIS
LIN {X 111.3156,Y -81.7391,Z 174,A -33.432,B 7.7849,C 0.329,E1 7.9219,E2 485.1679} C_DIS
LIN {X 113.8492,Y -78.1716,Z 174,A -31.6261,B 7.7851,C 0.3248,E1 7.9247,E2 483.3614} C_DIS
LIN {X 116.1827,Y -74.6598,Z 174,A -29.8936,B 7.7852,C 0.3209,E1 7.9274,E2 481.6294} C_DIS
LIN {X 118.6352,Y -70.6974,Z 174,A -28.0055,B 7.7854,C 0.3169,E1 7.9301,E2 479.7452} C_DIS
LIN {X 120.7887,Y -66.9517,Z 174,A -26.2425,B 7.7855,C 0.3129,E1 7.9325,E2 477.9843} C_DIS
LIN {X 123.1866,Y -62.4261,Z 174,A -24.1983,B 7.7857,C 0.309,E1 7.9352,E2 475.9484} C_DIS
LIN {X 126.4305,Y -55.5691,Z 174,A -21.1486,B 7.7859,C 0.3027,E1 7.9387,E2 472.9084} C_DIS
LIN {X 128.0379,Y -51.7514,Z 174,A -19.1525,B 7.7863,C 0.2924,E1 7.9409,E2 470.8745} C_DIS
LIN {X 129.264,Y -48.6083,Z 174,A -18.3195,B 7.786,C 0.3001,E1 7.9417,E2 470.1134} C_DIS
LIN {X 130.5829,Y -44.9458,Z 174,A -16.4899,B 7.7864,C 0.2913,E1 7.9434,E2 468.2545} C_DIS
LIN {X 131.732,Y -41.4604,Z 174,A -14.5054,B 7.7869,C 0.2776,E1 7.9451,E2 466.2087} C_DIS
LIN {X 132.9701,Y -37.2951,Z 174,A -13.1956,B 7.7867,C 0.2827,E1 7.9461,E2 464.961} C_DIS
LIN {X 134.032,Y -33.285,Z 174,A -11.5341,B 7.7868,C 0.2791,E1 7.9472,E2 463.3057} C_DIS
LIN {X 134.8398,Y -29.8447,Z 174,A -10.0633,B 7.787,C 0.2748,E1 7.9481,E2 461.8328} C_DIS
LIN {X 135.8403,Y -24.8945,Z 174,A -7.0678,B 7.7878,C 0.2503,E1 7.9497,E2 458.7185} C_DIS
LIN {X 136.932,Y -17.9345,Z 174,A -5.1962,B 7.7874,C 0.2636,E1 7.9504,E2 456.9805} C_DIS
LIN {X 137.7575,Y -9.7468,Z 174,A -1.098,B 7.7881,C 0.2397,E1 7.9514,E2 452.791} C_DIS
LIN {X 138.0419,Y -4.0666,Z 174,A 0.276,B 7.7877,C 0.2532,E1 7.9515,E2 451.5419} C_DIS
LIN {X 138.0323,Y 4.4123,Z 174,A 4.7194,B 7.7886,C 0.224,E1 7.9514,E2 446.9765} C_DIS
LIN {X 137.7162,Y 10.3126,Z 174,A 6.3399,B 7.7883,C 0.2341,E1 7.9511,E2 445.461} C_DIS
LIN {X 137.121,Y 16.4268,Z 174,A 8.5326,B 7.7883,C 0.2341,E1 7.9505,E2 443.3118} C_DIS
LIN {X 136.862,Y 18.4679,Z 174,A 9.8401,B 7.7886,C 0.2224,E1 7.95,E2 441.9457} C_DIS
LIN {X 136.2121,Y 22.7651,Z 174,A 11.5022,B 7.7886,C 0.2201,E1 7.9493,E2 440.3002} C_DIS
LIN {X 135.4784,Y 26.7985,Z 174,A 13.3843,B 7.7889,C 0.2116,E1 7.9483,E2 438.3937} C_DIS
LIN {X 134.5851,Y 30.9656,Z 174,A 14.8863,B 7.7889,C 0.2121,E1 7.9474,E2 436.9243} C_DIS
LIN {X 133.7969,Y 34.2111,Z 174,A 16.2732,B 7.789,C 0.2082,E1 7.9464,E2 435.5363} C_DIS
LIN {X 132.6312,Y 38.4839,Z 174,A 18.1237,B 7.7892,C 0.2029,E1 7.945,E2 433.6828} C_DIS
LIN {X 131.5029,Y 42.1776,Z 174,A 19.6197,B 7.7892,C 0.2006,E1 7.9438,E2 432.1992} C_DIS
LIN {X 130.4205,Y 45.4143,Z 174,A 21.0216,B 7.7893,C 0.197,E1 7.9425,E2 430.798} C_DIS
LIN {X 129.1718,Y 48.8545,Z 174,A 22.5272,B 7.7894,C 0.1932,E1 7.9411,E2 429.2932} C_DIS
LIN {X 127.2684,Y 53.6176,Z 174,A 24.5854,B 7.7895,C 0.189,E1 7.9389,E2 427.2425} C_DIS
LIN {X 125.9578,Y 56.6269,Z 174,A 25.9329,B 7.7895,C 0.1857,E1 7.9374,E2 425.896} C_DIS
LIN {X 124.4393,Y 59.8907,Z 174,A 27.4215,B 7.7897,C 0.1819,E1 7.9356,E2 424.4071} C_DIS
LIN {X 122.9173,Y 62.9551,Z 174,A 28.8298,B 7.7897,C 0.1785,E1 7.9338,E2 422.9994} C_DIS
LIN {X 120.9654,Y 66.6327,Z 174,A 31.4463,B 7.7902,C 0.1564,E1 7.9302,E2 420.2685} C_DIS
LIN {X 117.4491,Y 72.6519,Z 174,A 33.1671,B 7.7899,C 0.1727,E1 7.9279,E2 418.6956} C_DIS
LIN {X 114.3881,Y 77.381,Z 174,A 35.6976,B 7.7901,C 0.1632,E1 7.924,E2 416.1396} C_DIS
LIN {X 112.0317,Y 80.7557,Z 174,A 37.4581,B 7.7901,C 0.1582,E1 7.9211,E2 414.3717} C_DIS
LIN {X 108.8696,Y 84.9707,Z 174,A 39.3663,B 7.7901,C 0.1587,E1 7.9179,E2 412.4976} C_DIS
LIN {X 106.8465,Y 87.5003,Z 174,A 40.8974,B 7.7903,C 0.152,E1 7.9152,E2 410.9424} C_DIS
LIN {X 104.1617,Y 90.6797,Z 174,A 42.6064,B 7.7903,C 0.1486,E1 7.9121,E2 409.235} C_DIS
LIN {X 98.295,Y 97.0089,Z 174,A 45.9869,B 7.7904,C 0.1451,E1 7.9057,E2 405.8787} C_DIS
LIN {X 95.0212,Y 100.2175,Z 174,A 47.7329,B 7.7904,C 0.1443,E1 7.9022,E2 404.1517} C_DIS
LIN {X 93.019,Y 102.0784,Z 174,A 49.1121,B 7.7906,C 0.1374,E1 7.8993,E2 402.7415} C_DIS
LIN {X 90.6704,Y 104.1699,Z 174,A 50.3812,B 7.7906,C 0.1356,E1 7.8966,E2 401.4765} C_DIS
LIN {X 87.4726,Y 106.8691,Z 174,A 52.1365,B 7.7906,C 0.1321,E1 7.8929,E2 399.7185} C_DIS
LIN {X 83.9315,Y 109.672,Z 174,A 53.99,B 7.7907,C 0.1291,E1 7.8888,E2 397.8672} C_DIS
LIN {X 80.1688,Y 112.452,Z 174,A 56.6325,B 7.791,C 0.1126,E1 7.8826,E2 395.1357} C_DIS
LIN {X 75.0347,Y 115.9409,Z 174,A 58.2639,B 7.7908,C 0.1264,E1 7.8791,E2 393.6233} C_DIS
LIN {X 71.5182,Y 118.1423,Z 174,A 59.9308,B 7.7908,C 0.1248,E1 7.8751,E2 391.963} C_DIS
LIN {X 68.8161,Y 119.7372,Z 174,A 61.474,B 7.7908,C 0.1184,E1 7.8713,E2 390.3896} C_DIS
LIN {X 64.9043,Y 121.9014,Z 174,A 63.7397,B 7.791,C 0.1083,E1 7.8656,E2 388.0722} C_DIS
LIN {X 60.8292,Y 123.983,Z 174,A 65.1043,B 7.791,C 0.1157,E1 7.8624,E2 386.7747} C_DIS
LIN {X 57.324,Y 125.6437,Z 174,A 66.7282,B 7.791,C 0.1135,E1 7.8582,E2 385.1491} C_DIS
LIN {X 53.3646,Y 127.3741,Z 174,A 68.5378,B 7.791,C 0.1112,E1 7.8536,E2 383.3375} C_DIS
LIN {X 50.0365,Y 128.7178,Z 174,A 69.9285,B 7.791,C 0.1114,E1 7.85,E2 381.9591} C_DIS
LIN {X 46.7026,Y 129.9647,Z 174,A 71.3995,B 7.791,C 0.11,E1 7.8462,E2 380.4891} C_DIS
LIN {X 43.5809,Y 131.0444,Z 174,A 72.7585,B 7.791,C 0.109,E1 7.8426,E2 379.1317} C_DIS
LIN {X 40.3816,Y 132.0654,Z 174,A 74.1668,B 7.791,C 0.1075,E1 7.8388,E2 377.7218} C_DIS
LIN {X 37.3459,Y 132.9558,Z 174,A 75.5038,B 7.791,C 0.1061,E1 7.8352,E2 376.382} C_DIS
LIN {X 34.111,Y 133.8223,Z 174,A 76.8468,B 7.791,C 0.1059,E1 7.8316,E2 375.0451} C_DIS
LIN {X 28.4441,Y 135.1422,Z 174,A 79.1975,B 7.791,C 0.1055,E1 7.8252,E2 372.703} C_DIS
LIN {X 25.6424,Y 135.7002,Z 174,A 80.3855,B 7.791,C 0.1048,E1 7.822,E2 371.5149} C_DIS
LIN {X 22.477,Y 136.2602,Z 174,A 82.3612,B 7.7912,C 0.0929,E1 7.8163,E2 369.4592} C_DIS
LIN {X 17.4683,Y 136.993,Z 174,A 83.9607,B 7.7912,C 0.1009,E1 7.812,E2 367.9233} C_DIS
LIN {X 10.8652,Y 137.6755,Z 174,A 86.5682,B 7.7912,C 0.1027,E1 7.8049,E2 365.3352} C_DIS
LIN {X 3.6169,Y 138.0544,Z 174,A 89.5292,B 7.7912,C 0.1032,E1 7.7966,E2 362.3817} C_DIS
LIN {X -2.4267,Y 138.0804,Z 174,A 92.138,B 7.7912,C 0.1015,E1 7.7893,E2 359.7616} C_DIS
LIN {X -10.9119,Y 137.6716,Z 174,A 95.5898,B 7.7912,C 0.1033,E1 7.7797,E2 356.3208} C_DIS
LIN {X -16.7388,Y 137.0838,Z 174,A 98.084,B 7.7912,C 0.103,E1 7.7728,E2 353.8199} C_DIS
LIN {X -22.8,Y 136.2063,Z 174,A 100.4838,B 7.7911,C 0.1064,E1 7.7662,E2 351.4391} C_DIS
LIN {X -25.584,Y 135.7113,Z 174,A 101.8327,B 7.7911,C 0.1042,E1 7.7624,E2 350.0691} C_DIS
LIN {X -29.1628,Y 134.987,Z 174,A 103.3517,B 7.7911,C 0.105,E1 7.7583,E2 348.5505} C_DIS
LIN {X -32.4078,Y 134.2449,Z 174,A 104.7119,B 7.7911,C 0.1063,E1 7.7546,E2 347.1938} C_DIS
LIN {X -35.8913,Y 133.3562,Z 174,A 106.2456,B 7.7911,C 0.1067,E1 7.7504,E2 345.6558} C_DIS
LIN {X -38.9732,Y 132.488,Z 174,A 107.5505,B 7.7911,C 0.1081,E1 7.7469,E2 344.3548} C_DIS
LIN {X -42.3641,Y 131.4433,Z 174,A 109.0568,B 7.7911,C 0.1089,E1 7.7429,E2 342.8452} C_DIS
LIN {X -48.3766,Y 129.3508,Z 174,A 111.3917,B 7.7909,C 0.1163,E1 7.7369,E2 340.5502} C_DIS
LIN {X -51.7366,Y 128.0439,Z 174,A 113.1836,B 7.7909,C 0.1132,E1 7.7321,E2 338.7227} C_DIS
LIN {X -54.8506,Y 126.7411,Z 174,A 114.5705,B 7.7909,C 0.115,E1 7.7286,E2 337.3386} C_DIS
LIN {X -57.983,Y 125.339,Z 174,A 116.0282,B 7.7909,C 0.1162,E1 7.7248,E2 335.8778} C_DIS
LIN {X -62.0211,Y 123.3928,Z 174,A 117.8579,B 7.7909,C 0.119,E1 7.7203,E2 334.0533} C_DIS
LIN {X -64.4791,Y 122.1246,Z 174,A 119.088,B 7.7909,C 0.1193,E1 7.7172,E2 332.8139} C_DIS
LIN {X -69.5799,Y 119.2949,Z 174,A 121.4757,B 7.7909,C 0.1233,E1 7.7114,E2 330.4323} C_DIS
LIN {X -72.7028,Y 117.4174,Z 174,A 123.1511,B 7.7909,C 0.1231,E1 7.7074,E2 328.7379} C_DIS
LIN {X -76.3957,Y 115.049,Z 174,A 125.0064,B 7.7908,C 0.1254,E1 7.703,E2 326.8797} C_DIS
LIN {X -80.0888,Y 112.5092,Z 174,A 126.8803,B 7.7908,C 0.1283,E1 7.6987,E2 325.0056} C_DIS
LIN {X -84.6531,Y 109.116,Z 174,A 129.0455,B 7.7906,C 0.1353,E1 7.694,E2 322.8667} C_DIS
LIN {X -87.4834,Y 106.8603,Z 174,A 130.7618,B 7.7906,C 0.1349,E1 7.6902,E2 321.1251} C_DIS
LIN {X -91.0537,Y 103.8354,Z 174,A 132.7753,B 7.7906,C 0.1375,E1 7.6859,E2 319.1043} C_DIS
LIN {X -94.6178,Y 100.598,Z 174,A 134.7386,B 7.7906,C 0.1419,E1 7.6819,E2 317.1472} C_DIS
LIN {X -97.754,Y 97.5535,Z 174,A 136.5924,B 7.7904,C 0.145,E1 7.6782,E2 315.29} C_DIS
LIN {X -100.8598,Y 94.3389,Z 174,A 138.5264,B 7.7904,C 0.1478,E1 7.6745,E2 313.3479} C_DIS
LIN {X -103.8061,Y 91.0872,Z 174,A 140.3404,B 7.7904,C 0.1518,E1 7.6711,E2 311.5364} C_DIS
LIN {X -106.6828,Y 87.7006,Z 174,A 142.2226,B 7.7903,C 0.1553,E1 7.6677,E2 309.6512} C_DIS
LIN {X -111.1708,Y 81.9362,Z 174,A 145.0903,B 7.7901,C 0.1647,E1 7.6629,E2 306.8068} C_DIS
LIN {X -113.2143,Y 79.0887,Z 174,A 146.7273,B 7.7901,C 0.1655,E1 7.6602,E2 305.1484} C_DIS
LIN {X -115.5976,Y 75.5634,Z 174,A 148.6218,B 7.79,C 0.1679,E1 7.6573,E2 303.2395} C_DIS
LIN {X -117.8268,Y 72.037,Z 174,A 150.2809,B 7.7899,C 0.1732,E1 7.6549,E2 301.5911} C_DIS
LIN {X -120.0128,Y 68.3329,Z 174,A 152.0778,B 7.7898,C 0.1775,E1 7.6523,E2 299.7944} C_DIS
LIN {X -121.9726,Y 64.7686,Z 174,A 153.8253,B 7.7898,C 0.181,E1 7.65,E2 298.041} C_DIS
LIN {X -123.8625,Y 61.0735,Z 174,A 155.5262,B 7.7896,C 0.1857,E1 7.6479,E2 296.3443} C_DIS
LIN {X -125.4991,Y 57.6367,Z 174,A 157.1232,B 7.7895,C 0.1896,E1 7.646,E2 294.7468} C_DIS
LIN {X -126.8902,Y 54.5059,Z 174,A 158.5155,B 7.7894,C 0.1938,E1 7.6445,E2 293.3594} C_DIS
LIN {X -128.1171,Y 51.555,Z 174,A 159.8937,B 7.7894,C 0.1966,E1 7.643,E2 291.976} C_DIS
LIN {X -129.4162,Y 48.2021,Z 174,A 161.3756,B 7.7892,C 0.2008,E1 7.6415,E2 290.4968} C_DIS
LIN {X -130.5227,Y 45.1196,Z 174,A 162.7863,B 7.7892,C 0.2038,E1 7.6402,E2 289.0808} C_DIS
LIN {X -131.5815,Y 41.9314,Z 174,A 164.1857,B 7.789,C 0.2075,E1 7.639,E2 287.6821} C_DIS
LIN {X -132.5735,Y 38.6811,Z 174,A 165.6529,B 7.789,C 0.2106,E1 7.6378,E2 286.2091} C_DIS
LIN {X -133.4494,Y 35.5418,Z 174,A 167.0383,B 7.7889,C 0.214,E1 7.6368,E2 284.8208} C_DIS
LIN {X -134.2567,Y 32.359,Z 174,A 168.4511,B 7.7888,C 0.2171,E1 7.6359,E2 283.403} C_DIS
LIN {X -135.1185,Y 28.554,Z 174,A 170.3543,B 7.7888,C 0.2177,E1 7.6347,E2 281.4655} C_DIS
LIN {X -135.7605,Y 25.3266,Z 174,A 171.5786,B 7.7886,C 0.2235,E1 7.6341,E2 280.2603} C_DIS
LIN {X -136.4443,Y 21.3306,Z 174,A 173.1873,B 7.7884,C 0.2293,E1 7.6334,E2 278.6623} C_DIS
LIN {X -136.9597,Y 17.7228,Z 174,A 174.7074,B 7.7884,C 0.2336,E1 7.6328,E2 277.1427} C_DIS
LIN {X -137.4477,Y 13.4243,Z 174,A 176.6549,B 7.7882,C 0.2366,E1 7.6322,E2 275.1775} C_DIS
LIN {X -137.7796,Y 9.4441,Z 174,A 178.3054,B 7.7881,C 0.2414,E1 7.6319,E2 273.5294} C_DIS
LIN {X -137.9943,Y 5.4414,Z 174,A 179.921,B 7.7879,C 0.2469,E1 7.6317,E2 271.9212} C_DIS
LIN {X -138.0915,Y 1.758,Z 174,A -178.3506,B 7.7879,C 0.2485,E1 7.6316,E2 270.169} C_DIS
LIN {X -138.0707,Y -3.005,Z 174,A -176.5462,B 7.7876,C 0.2566,E1 7.6316,E2 268.388} C_DIS
LIN {X -137.9585,Y -6.3147,Z 174,A -174.9978,B 7.7876,C 0.2581,E1 7.6318,E2 266.8187} C_DIS
LIN {X -137.7145,Y -10.335,Z 174,A -173.404,B 7.7873,C 0.264,E1 7.6321,E2 265.236} C_DIS
LIN {X -137.3159,Y -14.7092,Z 174,A -171.672,B 7.7871,C 0.2705,E1 7.6326,E2 263.5171} C_DIS
LIN {X -136.9506,Y -17.792,Z 174,A -170.1826,B 7.7871,C 0.2713,E1 7.6331,E2 262.0032} C_DIS
LIN {X -136.3602,Y -21.8737,Z 174,A -168.3525,B 7.787,C 0.2745,E1 7.6339,E2 260.1594} C_DIS
LIN {X -135.6156,Y -26.0845,Z 174,A -166.7192,B 7.7867,C 0.2815,E1 7.6347,E2 258.5453} C_DIS
LIN {X -134.9733,Y -29.2264,Z 174,A -165.314,B 7.7867,C 0.2842,E1 7.6355,E2 257.1316} C_DIS
LIN {X -134.1983,Y -32.601,Z 174,A -163.8301,B 7.7865,C 0.2875,E1 7.6365,E2 255.6428} C_DIS
LIN {X -133.3521,Y -35.9064,Z 174,A -162.4532,B 7.7864,C 0.292,E1 7.6375,E2 254.2718} C_DIS
LIN {X -132.4511,Y -39.099,Z 174,A -161.0297,B 7.7862,C 0.2951,E1 7.6386,E2 252.8433} C_DIS
LIN {X -131.4812,Y -42.2455,Z 174,A -159.6459,B 7.7862,C 0.2985,E1 7.6397,E2 251.4581} C_DIS
LIN {X -130.1135,Y -46.2899,Z 174,A -157.9298,B 7.7859,C 0.3041,E1 7.6413,E2 249.7504} C_DIS
LIN {X -128.3543,Y -50.9667,Z 174,A -155.7704,B 7.7857,C 0.3084,E1 7.6435,E2 247.5814} C_DIS
LIN {X -127.2837,Y -53.5809,Z 174,A -154.504,B 7.7857,C 0.3101,E1 7.6448,E2 246.3036} C_DIS
LIN {X -125.8843,Y -56.7911,Z 174,A -153.0283,B 7.7855,C 0.3136,E1 7.6465,E2 244.8259} C_DIS
LIN {X -124.4983,Y -59.7674,Z 174,A -151.6513,B 7.7854,C 0.3168,E1 7.6481,E2 243.4477} C_DIS
LIN {X -122.7674,Y -63.2494,Z 174,A -149.7028,B 7.7854,C 0.316,E1 7.6507,E2 241.4574} C_DIS
LIN {X -121.1458,Y -66.3038,Z 174,A -148.5586,B 7.7851,C 0.3239,E1 7.6521,E2 240.3512} C_DIS
LIN {X -119.2451,Y -69.6647,Z 174,A -146.8368,B 7.7851,C 0.326,E1 7.6546,E2 238.6149} C_DIS
LIN {X -117.0144,Y -73.3503,Z 174,A -144.9903,B 7.7849,C 0.3295,E1 7.6573,E2 236.7617} C_DIS
LIN {X -114.5825,Y -77.0937,Z 174,A -143.2279,B 7.7846,C 0.3351,E1 7.66,E2 235.0117} C_DIS
LIN {X -112.2827,Y -80.4055,Z 174,A -141.4583,B 7.7846,C 0.3376,E1 7.6628,E2 233.2304} C_DIS
LIN {X -109.5803,Y -84.0514,Z 174,A -139.5613,B 7.7843,C 0.3416,E1 7.666,E2 231.3324} C_DIS
LIN {X -106.9578,Y -87.3641,Z 174,A -137.7689,B 7.7843,C 0.3448,E1 7.6692,E2 229.5356} C_DIS
LIN {X -104.0697,Y -90.7852,Z 174,A -135.6447,B 7.7843,C 0.3447,E1 7.6731,E2 227.3777} C_DIS
LIN {X -101.7765,Y -93.3488,Z 174,A -134.4246,B 7.7839,C 0.3508,E1 7.6754,E2 226.1847} C_DIS
LIN {X -98.6761,Y -96.6203,Z 174,A -132.514,B 7.7838,C 0.3539,E1 7.6791,E2 224.2695} C_DIS
LIN {X -96.3055,Y -98.9839,Z 174,A -131.1104,B 7.7837,C 0.3564,E1 7.6819,E2 222.8645} C_DIS
LIN {X -93.0906,Y -102.0134,Z 174,A -129.2512,B 7.7835,C 0.3594,E1 7.6857,E2 221.0023} C_DIS
LIN {X -89.7338,Y -104.9783,Z 174,A -127.365,B 7.7835,C 0.3624,E1 7.6897,E2 219.1129} C_DIS
LIN {X -86.2738,Y -107.8397,Z 174,A -125.4621,B 7.7833,C 0.365,E1 7.6938,E2 217.2052} C_DIS
LIN {X -82.5791,Y -110.694,Z 174,A -123.2176,B 7.7833,C 0.3633,E1 7.6989,E2 214.9211} C_DIS
LIN {X -79.3397,Y -113.0388,Z 174,A -121.8661,B 7.783,C 0.3708,E1 7.7019,E2 213.6098} C_DIS
LIN {X -75.6164,Y -115.5628,Z 174,A -119.8859,B 7.783,C 0.3718,E1 7.7065,E2 211.615} C_DIS
LIN {X -71.2965,Y -118.2763,Z 174,A -117.8552,B 7.7828,C 0.3761,E1 7.7113,E2 209.5955} C_DIS
LIN {X -67.4448,Y -120.5144,Z 174,A -115.643,B 7.7829,C 0.3727,E1 7.7168,E2 207.3361} C_DIS
LIN {X -64.0159,Y -122.3678,Z 174,A -114.4213,B 7.7825,C 0.3811,E1 7.7197,E2 206.1656} C_DIS
LIN {X -60.509,Y -124.141,Z 174,A -112.8128,B 7.7825,C 0.3834,E1 7.7237,E2 204.56} C_DIS
LIN {X -57.2117,Y -125.6954,Z 174,A -111.2828,B 7.7823,C 0.3848,E1 7.7276,E2 203.0277} C_DIS
LIN {X -53.9412,Y -127.1332,Z 174,A -109.8146,B 7.7823,C 0.3866,E1 7.7314,E2 201.5611} C_DIS
LIN {X -49.894,Y -128.7731,Z 174,A -107.9782,B 7.7822,C 0.3879,E1 7.7362,E2 199.7212} C_DIS
LIN {X -46.6549,Y -129.9819,Z 174,A -106.5288,B 7.7822,C 0.3889,E1 7.74,E2 198.2697} C_DIS
LIN {X -43.3583,Y -131.1185,Z 174,A -104.9957,B 7.7822,C 0.3886,E1 7.7441,E2 196.7252} C_DIS
LIN {X -39.219,Y -132.416,Z 174,A -103.231,B 7.7821,C 0.3905,E1 7.7488,E2 194.9648} C_DIS
LIN {X -35.7422,Y -133.3959,Z 174,A -101.1465,B 7.7825,C 0.3816,E1 7.7546,E2 192.8034} C_DIS
LIN {X -30.8886,Y -134.6027,Z 174,A -99.701,B 7.7819,C 0.3934,E1 7.7583,E2 191.4396} C_DIS
LIN {X -27.4792,Y -135.3398,Z 174,A -98.2438,B 7.7819,C 0.3939,E1 7.7623,E2 189.9807} C_DIS
LIN {X -21.9665,Y -136.3445,Z 174,A -95.9314,B 7.7819,C 0.3951,E1 7.7687,E2 187.6693} C_DIS
LIN {X -17.157,Y -137.0338,Z 174,A -93.8904,B 7.7819,C 0.3951,E1 7.7743,E2 185.6244} C_DIS
LIN {X -13.0467,Y -137.4839,Z 174,A -92.1094,B 7.7819,C 0.3943,E1 7.7793,E2 183.8341} C_DIS
LIN {X -8.8214,Y -137.8199,Z 174,A -90.3572,B 7.7819,C 0.3946,E1 7.7842,E2 182.082} C_DIS
LIN {X -4.7273,Y -138.0222,Z 174,A -88.5428,B 7.7819,C 0.3926,E1 7.7893,E2 180.2521} C_DIS
LIN {X -0.5963,Y -138.1004,Z 174,A -86.9233,B 7.7819,C 0.3941,E1 7.7938,E2 178.6441} C_DIS
LIN {X -0.5963,Y -138.1004,Z 174,A -86.9233,B 7.7819,C 0.3941,E1 7.7938,E2 178.6441} C_DIS
Enddeposition()
LIN {X 0.9845,Y -139.0008,Z 174,A -86.667,B 7.7645,C 0.4057,E1 7.7774,E2 178.4776} C_DIS
Startdeposition()
$VEL.CP = VEL_PRINT
LIN {X -2.1074,Y -138.9929,Z 174,A -88.1967,B 7.7642,C 0.4104,E1 7.7731,E2 180.0412} C_DIS
LIN {X -5.6232,Y -138.8951,Z 174,A -89.6963,B 7.7642,C 0.4113,E1 7.7689,E2 181.5479} C_DIS
LIN {X -10.0005,Y -138.6485,Z 174,A -91.4545,B 7.7642,C 0.4103,E1 7.764,E2 183.3006} C_DIS
LIN {X -13.3305,Y -138.368,Z 174,A -92.8022,B 7.7642,C 0.4096,E1 7.7602,E2 184.645} C_DIS
LIN {X -16.5409,Y -138.021,Z 174,A -94.1266,B 7.7642,C 0.4092,E1 7.7566,E2 185.9689} C_DIS
LIN {X -21.4379,Y -137.3456,Z 174,A -96.8362,B 7.7637,C 0.42,E1 7.7488,E2 188.7659} C_DIS
LIN {X -26.596,Y -136.4414,Z 174,A -98.2817,B 7.7644,C 0.4071,E1 7.7451,E2 190.1203} C_DIS
LIN {X -32.3669,Y -135.1879,Z 174,A -101.2856,B 7.764,C 0.4154,E1 7.7367,E2 193.1983} C_DIS
LIN {X -36.6864,Y -134.0822,Z 174,A -102.7771,B 7.7643,C 0.4085,E1 7.7328,E2 194.6457} C_DIS
LIN {X -40.3925,Y -133.0107,Z 174,A -104.2378,B 7.7645,C 0.4052,E1 7.729,E2 196.0899} C_DIS
LIN {X -43.6076,Y -131.9916,Z 174,A -105.6504,B 7.7645,C 0.4045,E1 7.7252,E2 197.5057} C_DIS
LIN {X -46.8729,Y -130.8675,Z 174,A -107.021,B 7.7647,C 0.4024,E1 7.7216,E2 198.8697} C_DIS
LIN {X -50.0884,Y -129.6708,Z 174,A -108.5324,B 7.7647,C 0.4027,E1 7.7176,E2 200.3938} C_DIS
LIN {X -53.408,Y -128.339,Z 174,A -109.99,B 7.7647,C 0.401,E1 7.7139,E2 201.8494} C_DIS
LIN {X -57.6692,Y -126.4835,Z 174,A -112.0287,B 7.7647,C 0.401,E1 7.7086,E2 203.9042} C_DIS
LIN {X -61.7442,Y -124.5431,Z 174,A -114.7579,B 7.7641,C 0.4127,E1 7.7015,E2 206.7445} C_DIS
LIN {X -67.9836,Y -121.2521,Z 174,A -116.8181,B 7.765,C 0.3955,E1 7.6967,E2 208.6966} C_DIS
LIN {X -71.9652,Y -118.9321,Z 174,A -118.729,B 7.7651,C 0.3931,E1 7.6921,E2 210.6089} C_DIS
LIN {X -77.3139,Y -115.5267,Z 174,A -122.2414,B 7.7646,C 0.4032,E1 7.6837,E2 214.2357} C_DIS
LIN {X -82.9847,Y -111.5229,Z 174,A -124.2608,B 7.7655,C 0.3856,E1 7.6794,E2 216.1475} C_DIS
LIN {X -86.6116,Y -108.7302,Z 174,A -126.1358,B 7.7657,C 0.3822,E1 7.6753,E2 218.0206} C_DIS
LIN {X -90.0161,Y -105.9289,Z 174,A -128.0074,B 7.7657,C 0.3799,E1 7.6712,E2 219.8989} C_DIS
LIN {X -93.5269,Y -102.8424,Z 174,A -129.9079,B 7.766,C 0.3759,E1 7.6673,E2 221.7955} C_DIS
LIN {X -96.9916,Y -99.5822,Z 174,A -132.252,B 7.7659,C 0.378,E1 7.6625,E2 224.1881} C_DIS
LIN {X -99.7181,Y -96.8513,Z 174,A -133.5342,B 7.7662,C 0.3702,E1 7.66,E2 225.4305} C_DIS
LIN {X -105.0069,Y -91.0908,Z 174,A -136.848,B 7.7665,C 0.3649,E1 7.6538,E2 228.7548} C_DIS
LIN {X -107.9037,Y -87.6401,Z 174,A -138.7306,B 7.7667,C 0.3612,E1 7.6505,E2 230.64} C_DIS
LIN {X -110.5988,Y -84.213,Z 174,A -140.4838,B 7.7669,C 0.3566,E1 7.6475,E2 232.3868} C_DIS
LIN {X -113.2037,Y -80.677,Z 174,A -142.3229,B 7.767,C 0.3529,E1 7.6444,E2 234.2288} C_DIS
LIN {X -115.6491,Y -77.1305,Z 174,A -144.2351,B 7.7671,C 0.3508,E1 7.6414,E2 236.1575} C_DIS
LIN {X -118.2312,Y -73.112,Z 174,A -146.1969,B 7.7674,C 0.346,E1 7.6385,E2 238.1175} C_DIS
LIN {X -120.4753,Y -69.3516,Z 174,A -148.102,B 7.7674,C 0.343,E1 7.6358,E2 240.0344} C_DIS
LIN {X -123.5219,Y -63.7669,Z 174,A -150.6786,B 7.7678,C 0.3358,E1 7.6324,E2 242.6038} C_DIS
LIN {X -125.2367,Y -60.326,Z 174,A -152.2505,B 7.768,C 0.3316,E1 7.6305,E2 244.1731} C_DIS
LIN {X -126.8014,Y -56.9625,Z 174,A -153.7571,B 7.7682,C 0.3273,E1 7.6287,E2 245.6759} C_DIS
LIN {X -128.1856,Y -53.7754,Z 174,A -155.1991,B 7.7683,C 0.3237,E1 7.6272,E2 247.1183} C_DIS
LIN {X -129.9684,Y -49.3139,Z 174,A -157.8027,B 7.7682,C 0.3273,E1 7.6245,E2 249.7993} C_DIS
LIN {X -131.633,Y -44.6845,Z 174,A -159.4182,B 7.7686,C 0.316,E1 7.623,E2 251.3615} C_DIS
LIN {X -132.8637,Y -40.8729,Z 174,A -160.9481,B 7.7689,C 0.3098,E1 7.6218,E2 252.8749} C_DIS
LIN {X -133.8355,Y -37.5685,Z 174,A -162.3917,B 7.769,C 0.3062,E1 7.6206,E2 254.3206} C_DIS
LIN {X -134.6501,Y -34.5372,Z 174,A -163.6553,B 7.7692,C 0.3022,E1 7.6198,E2 255.5794} C_DIS
LIN {X -135.4073,Y -31.4396,Z 174,A -165.1272,B 7.7692,C 0.3008,E1 7.6188,E2 257.0703} C_DIS
LIN {X -136.2075,Y -27.7644,Z 174,A -166.6456,B 7.7694,C 0.296,E1 7.6179,E2 258.5834} C_DIS
LIN {X -136.9156,Y -24.0352,Z 174,A -168.3711,B 7.7694,C 0.2938,E1 7.617,E2 260.328} C_DIS
LIN {X -137.5592,Y -20.0244,Z 174,A -170.0047,B 7.7697,C 0.2885,E1 7.6164,E2 261.9551} C_DIS
LIN {X -138.054,Y -16.2643,Z 174,A -172.1044,B 7.7696,C 0.2915,E1 7.6157,E2 264.121} C_DIS
LIN {X -138.5289,Y -11.5398,Z 174,A -173.5929,B 7.77,C 0.2794,E1 7.6153,E2 265.549} C_DIS
LIN {X -138.8273,Y -7.0992,Z 174,A -175.1636,B 7.7703,C 0.2704,E1 7.615,E2 267.085} C_DIS
LIN {X -138.9269,Y -4.8075,Z 174,A -176.5708,B 7.7703,C 0.2741,E1 7.6149,E2 268.5496} C_DIS
LIN {X -138.9902,Y 2.2686,Z 174,A -179.3469,B 7.7706,C 0.2638,E1 7.6149,E2 271.3055} C_DIS
LIN {X -138.8733,Y 6.1812,Z 174,A 179.0464,B 7.7707,C 0.2591,E1 7.615,E2 272.9099} C_DIS
LIN {X -138.7067,Y 9.1792,Z 174,A 177.4987,B 7.7707,C 0.2598,E1 7.6153,E2 274.4954} C_DIS
LIN {X -138.0831,Y 16.0199,Z 174,A 174.8134,B 7.771,C 0.2496,E1 7.616,E2 277.1598} C_DIS
LIN {X -137.6516,Y 19.3774,Z 174,A 173.4955,B 7.7712,C 0.2446,E1 7.6165,E2 278.4667} C_DIS
LIN {X -137.0179,Y 23.4474,Z 174,A 170.9817,B 7.771,C 0.251,E1 7.6178,E2 281.0806} C_DIS
LIN {X -135.9602,Y 28.9539,Z 174,A 169.4177,B 7.7715,C 0.2341,E1 7.6186,E2 282.5495} C_DIS
LIN {X -135.183,Y 32.3871,Z 174,A 167.8974,B 7.7715,C 0.231,E1 7.6195,E2 284.0771} C_DIS
LIN {X -134.3398,Y 35.7234,Z 174,A 166.4398,B 7.7717,C 0.2276,E1 7.6205,E2 285.5383} C_DIS
LIN {X -133.527,Y 38.6529,Z 174,A 165.1272,B 7.7717,C 0.2249,E1 7.6216,E2 286.857} C_DIS
LIN {X -132.5789,Y 41.7902,Z 174,A 163.8096,B 7.7719,C 0.2207,E1 7.6226,E2 288.1692} C_DIS
LIN {X -131.4815,Y 45.1231,Z 174,A 162.2147,B 7.7719,C 0.2188,E1 7.6241,E2 289.7813} C_DIS
LIN {X -130.2396,Y 48.5897,Z 174,A 160.8271,B 7.7721,C 0.2129,E1 7.6254,E2 291.1511} C_DIS
LIN {X -129.0307,Y 51.7149,Z 174,A 159.3612,B 7.7721,C 0.2103,E1 7.6269,E2 292.6263} C_DIS
LIN {X -127.7747,Y 54.7459,Z 174,A 157.9439,B 7.7723,C 0.2076,E1 7.6284,E2 294.0503} C_DIS
LIN {X -126.356,Y 57.9449,Z 174,A 156.495,B 7.7723,C 0.2039,E1 7.6301,E2 295.4987} C_DIS
LIN {X -123.9592,Y 62.9079,Z 174,A 154.2172,B 7.7725,C 0.1981,E1 7.6329,E2 297.775} C_DIS
LIN {X -122.231,Y 66.2086,Z 174,A 152.4686,B 7.7725,C 0.1972,E1 7.6352,E2 299.5486} C_DIS
LIN {X -119.8004,Y 70.5103,Z 174,A 150.5146,B 7.7727,C 0.1909,E1 7.6379,E2 301.4904} C_DIS
LIN {X -116.5226,Y 75.8046,Z 174,A 147.8794,B 7.7728,C 0.1856,E1 7.6419,E2 304.1316} C_DIS
LIN {X -114.0145,Y 79.527,Z 174,A 145.9825,B 7.7728,C 0.1818,E1 7.6449,E2 306.0325} C_DIS
LIN {X -111.6924,Y 82.7571,Z 174,A 144.487,B 7.773,C 0.1759,E1 7.6473,E2 307.5085} C_DIS
LIN {X -108.5665,Y 86.8173,Z 174,A 142.1932,B 7.773,C 0.1737,E1 7.6513,E2 309.823} C_DIS
LIN {X -105.5057,Y 90.5121,Z 174,A 140.0279,B 7.7731,C 0.172,E1 7.6552,E2 312.0096} C_DIS
LIN {X -100.7218,Y 95.8073,Z 174,A 137.1572,B 7.7733,C 0.1647,E1 7.6606,E2 314.8687} C_DIS
LIN {X -97.57,Y 99.0153,Z 174,A 135.5086,B 7.7734,C 0.1579,E1 7.6638,E2 316.4902} C_DIS
LIN {X -93.8721,Y 102.5277,Z 174,A 132.9013,B 7.7734,C 0.1611,E1 7.6692,E2 319.158} C_DIS
LIN {X -91.0769,Y 105.019,Z 174,A 131.5783,B 7.7734,C 0.1549,E1 7.672,E2 320.4524} C_DIS
LIN {X -87.6322,Y 107.9102,Z 174,A 129.8858,B 7.7736,C 0.1491,E1 7.6756,E2 322.1234} C_DIS
LIN {X -82.0246,Y 112.2315,Z 174,A 126.7837,B 7.7736,C 0.1468,E1 7.6825,E2 325.2457} C_DIS
LIN {X -78.3698,Y 114.8134,Z 174,A 124.9179,B 7.7736,C 0.144,E1 7.6868,E2 327.1126} C_DIS
LIN {X -75.664,Y 116.6138,Z 174,A 123.3492,B 7.7736,C 0.1454,E1 7.6905,E2 328.7084} C_DIS
LIN {X -72.779,Y 118.4359,Z 174,A 121.2999,B 7.7736,C 0.1529,E1 7.6956,E2 330.8352} C_DIS
LIN {X -66.8866,Y 121.8612,Z 174,A 119.2908,B 7.7738,C 0.1368,E1 7.7003,E2 332.7441} C_DIS
LIN {X -63.4154,Y 123.7009,Z 174,A 117.7562,B 7.7738,C 0.1333,E1 7.704,E2 334.2668} C_DIS
LIN {X -57.6005,Y 126.5153,Z 174,A 114.949,B 7.7738,C 0.1323,E1 7.7111,E2 337.0899} C_DIS
LIN {X -53.9461,Y 128.1143,Z 174,A 113.4222,B 7.774,C 0.1286,E1 7.715,E2 338.6009} C_DIS
LIN {X -50.1197,Y 129.6587,Z 174,A 111.4325,B 7.774,C 0.1313,E1 7.7203,E2 340.6249} C_DIS
LIN {X -47.0817,Y 130.7923,Z 174,A 110.1928,B 7.774,C 0.1284,E1 7.7235,E2 341.8518} C_DIS
LIN {X -42.5304,Y 132.3425,Z 174,A 108.3663,B 7.774,C 0.1242,E1 7.7283,E2 343.6577} C_DIS
LIN {X -39.1783,Y 133.3731,Z 174,A 106.9334,B 7.774,C 0.1227,E1 7.7321,E2 345.0881} C_DIS
LIN {X -34.8619,Y 134.5676,Z 174,A 104.947,B 7.774,C 0.1236,E1 7.7375,E2 347.0907} C_DIS
LIN {X -31.4606,Y 135.4025,Z 174,A 103.6017,B 7.774,C 0.1211,E1 7.7411,E2 348.4229} C_DIS
LIN {X -28.1289,Y 136.1334,Z 174,A 102.2529,B 7.774,C 0.1193,E1 7.7448,E2 349.7638} C_DIS
LIN {X -24.5532,Y 136.8229,Z 174,A 100.6913,B 7.774,C 0.1195,E1 7.7491,E2 351.332} C_DIS
LIN {X -18.7564,Y 137.7391,Z 174,A 98.2092,B 7.774,C 0.1195,E1 7.756,E2 353.8206} C_DIS
LIN {X -11.0198,Y 138.5728,Z 174,A 95.0996,B 7.7741,C 0.1169,E1 7.7646,E2 356.9164} C_DIS
LIN {X -4.851,Y 138.9252,Z 174,A 92.4049,B 7.7741,C 0.119,E1 7.7721,E2 359.6282} C_DIS
LIN {X -1.1571,Y 139.0045,Z 174,A 91.0466,B 7.7741,C 0.1162,E1 7.7759,E2 360.9654} C_DIS
LIN {X 1.8577,Y 138.9971,Z 174,A 89.5847,B 7.7741,C 0.1199,E1 7.78,E2 362.4539} C_DIS
LIN {X 9.0713,Y 138.7134,Z 174,A 86.6865,B 7.7741,C 0.119,E1 7.7881,E2 365.3413} C_DIS
LIN {X 12.5293,Y 138.4449,Z 174,A 84.7647,B 7.774,C 0.1277,E1 7.7936,E2 367.3233} C_DIS
LIN {X 17.372,Y 137.9205,Z 174,A 83.4015,B 7.7741,C 0.1174,E1 7.7972,E2 368.6064} C_DIS
LIN {X 21.1497,Y 137.3902,Z 174,A 81.5859,B 7.7741,C 0.1222,E1 7.8023,E2 370.4515} C_DIS
LIN {X 25.7489,Y 136.6034,Z 174,A 78.7733,B 7.7738,C 0.1386,E1 7.8103,E2 373.3726} C_DIS
LIN {X 33.2692,Y 134.9704,Z 174,A 76.5664,B 7.774,C 0.1239,E1 7.816,E2 375.4606} C_DIS
LIN {X 37.2739,Y 133.9179,Z 174,A 75.0076,B 7.774,C 0.1226,E1 7.8201,E2 377.0005} C_DIS
LIN {X 40.5478,Y 132.9632,Z 174,A 73.6007,B 7.774,C 0.1237,E1 7.8239,E2 378.4074} C_DIS
LIN {X 43.8004,Y 131.9274,Z 174,A 72.1996,B 7.774,C 0.1249,E1 7.8276,E2 379.8075} C_DIS
LIN {X 46.9361,Y 130.8447,Z 174,A 70.8264,B 7.774,C 0.1263,E1 7.8312,E2 381.1813} C_DIS
LIN {X 50.1285,Y 129.6553,Z 174,A 69.4623,B 7.774,C 0.127,E1 7.8347,E2 382.5402} C_DIS
LIN {X 55.5393,Y 127.4317,Z 174,A 67.0148,B 7.774,C 0.1303,E1 7.8411,E2 384.9921} C_DIS
LIN {X 58.1762,Y 126.2491,Z 174,A 64.7382,B 7.7735,C 0.1513,E1 7.8472,E2 387.4023} C_DIS
LIN {X 65.3805,Y 122.6759,Z 174,A 62.4742,B 7.7738,C 0.1367,E1 7.8525,E2 389.5372} C_DIS
LIN {X 69.3389,Y 120.4827,Z 174,A 60.6049,B 7.7738,C 0.1394,E1 7.857,E2 391.407} C_DIS
LIN {X 72.6411,Y 118.5205,Z 174,A 59.0897,B 7.7738,C 0.1405,E1 7.8606,E2 392.9138} C_DIS
LIN {X 75.4319,Y 116.7645,Z 174,A 57.5626,B 7.7737,C 0.1457,E1 7.8642,E2 394.462} C_DIS
LIN {X 80.6514,Y 113.2221,Z 174,A 55.1325,B 7.7737,C 0.1467,E1 7.8698,E2 396.8712} C_DIS
LIN {X 84.3947,Y 110.4598,Z 174,A 53.2649,B 7.7736,C 0.1491,E1 7.8739,E2 398.7329} C_DIS
LIN {X 87.8524,Y 107.7302,Z 174,A 51.4669,B 7.7736,C 0.152,E1 7.8778,E2 400.5291} C_DIS
LIN {X 91.1443,Y 104.9602,Z 174,A 49.9975,B 7.7736,C 0.1495,E1 7.8809,E2 401.9609} C_DIS
LIN {X 93.4229,Y 102.9367,Z 174,A 48.6756,B 7.7736,C 0.1532,E1 7.8837,E2 403.2913} C_DIS
LIN {X 96.3588,Y 100.1932,Z 174,A 46.8107,B 7.7734,C 0.1604,E1 7.8875,E2 405.1827} C_DIS
LIN {X 99.5111,Y 97.0644,Z 174,A 44.2993,B 7.773,C 0.1772,E1 7.8926,E2 407.7794} C_DIS
LIN {X 103.8034,Y 92.4598,Z 174,A 42.4801,B 7.7732,C 0.1678,E1 7.8958,E2 409.503} C_DIS
LIN {X 106.779,Y 89.0071,Z 174,A 40.5917,B 7.7732,C 0.1721,E1 7.8992,E2 411.3934} C_DIS
LIN {X 111.0688,Y 83.5917,Z 174,A 37.8183,B 7.773,C 0.1771,E1 7.904,E2 414.1586} C_DIS
LIN {X 113.7117,Y 79.9594,Z 174,A 36.0205,B 7.773,C 0.1804,E1 7.9069,E2 415.9505} C_DIS
LIN {X 115.7708,Y 76.9481,Z 174,A 34.4927,B 7.7728,C 0.1844,E1 7.9093,E2 417.4821} C_DIS
LIN {X 117.6575,Y 74.031,Z 174,A 32.7752,B 7.7726,C 0.1935,E1 7.9119,E2 419.2361} C_DIS
LIN {X 119.7567,Y 70.5843,Z 174,A 31.1416,B 7.7726,C 0.197,E1 7.9142,E2 420.8669} C_DIS
LIN {X 121.7631,Y 67.0646,Z 174,A 29.8123,B 7.7726,C 0.1945,E1 7.9159,E2 422.1543} C_DIS
LIN {X 123.7227,Y 63.3725,Z 174,A 28.1964,B 7.7726,C 0.1967,E1 7.918,E2 423.7577} C_DIS
LIN {X 125.0788,Y 60.6565,Z 174,A 26.6794,B 7.7723,C 0.2052,E1 7.9199,E2 425.3089} C_DIS
LIN {X 126.5484,Y 57.5281,Z 174,A 25.5513,B 7.7723,C 0.2031,E1 7.9212,E2 426.4005} C_DIS
LIN {X 129.1177,Y 51.4991,Z 174,A 22.814,B 7.7722,C 0.2109,E1 7.9241,E2 429.1441} C_DIS
LIN {X 130.6761,Y 47.4039,Z 174,A 21.19,B 7.7722,C 0.2121,E1 7.9257,E2 430.7462} C_DIS
LIN {X 131.8152,Y 44.1374,Z 174,A 19.7554,B 7.772,C 0.2162,E1 7.927,E2 432.1829} C_DIS
LIN {X 132.8773,Y 40.8284,Z 174,A 18.348,B 7.772,C 0.2196,E1 7.9282,E2 433.5881} C_DIS
LIN {X 133.8404,Y 37.5509,Z 174,A 16.9898,B 7.7718,C 0.2225,E1 7.9292,E2 434.941} C_DIS
LIN {X 134.7695,Y 34.0667,Z 174,A 15.4796,B 7.7718,C 0.2271,E1 7.9303,E2 436.4553} C_DIS
LIN {X 135.4508,Y 31.2491,Z 174,A 13.7255,B 7.7713,C 0.2417,E1 7.9314,E2 438.2809} C_DIS
LIN {X 136.5053,Y 26.262,Z 174,A 12.2951,B 7.7715,C 0.2341,E1 7.9322,E2 439.6283} C_DIS
LIN {X 137.243,Y 22.0987,Z 174,A 10.322,B 7.7712,C 0.2437,E1 7.9331,E2 441.6321} C_DIS
LIN {X 137.816,Y 18.1696,Z 174,A 8.3131,B 7.7708,C 0.2559,E1 7.9338,E2 443.6893} C_DIS
LIN {X 138.4107,Y 12.8856,Z 174,A 6.6916,B 7.771,C 0.2507,E1 7.9343,E2 445.2405} C_DIS
LIN {X 138.7429,Y 8.5919,Z 174,A 4.5603,B 7.7706,C 0.263,E1 7.9347,E2 447.4185} C_DIS
LIN {X 138.949,Y 4.0814,Z 174,A 2.8372,B 7.7705,C 0.2656,E1 7.9347,E2 449.1258} C_DIS
LIN {X 139.0124,Y -0.0764,Z 174,A 1.4947,B 7.7705,C 0.263,E1 7.9348,E2 450.4226} C_DIS
LIN {X 138.9554,Y -3.8487,Z 174,A 0.0213,B 7.7705,C 0.2658,E1 7.9348,E2 451.8869} C_DIS
LIN {X 138.6229,Y -10.3507,Z 174,A -3.1699,B 7.7699,C 0.2839,E1 7.9342,E2 455.1451} C_DIS
LIN {X 138.1776,Y -15.1797,Z 174,A -4.589,B 7.7701,C 0.2778,E1 7.9338,E2 456.4923} C_DIS
LIN {X 137.6524,Y -19.3718,Z 174,A -6.0795,B 7.7701,C 0.2778,E1 7.9332,E2 457.9522} C_DIS
LIN {X 137.0469,Y -23.2737,Z 174,A -8.558,B 7.7693,C 0.2997,E1 7.9321,E2 460.5408} C_DIS
LIN {X 136.01,Y -28.7232,Z 174,A -10.196,B 7.7695,C 0.293,E1 7.9312,E2 462.0985} C_DIS
LIN {X 135.1864,Y -32.3729,Z 174,A -11.6195,B 7.7695,C 0.295,E1 7.9303,E2 463.5082} C_DIS
LIN {X 134.3675,Y -35.6194,Z 174,A -13.1691,B 7.7692,C 0.3023,E1 7.9292,E2 465.0809} C_DIS
LIN {X 132.5771,Y -41.796,Z 174,A -15.5391,B 7.7692,C 0.304,E1 7.9273,E2 467.4175} C_DIS
LIN {X 131.3728,Y -45.4369,Z 174,A -17.1074,B 7.7689,C 0.3081,E1 7.9259,E2 468.9857} C_DIS
LIN {X 130.348,Y -48.3003,Z 174,A -18.5431,B 7.7687,C 0.3152,E1 7.9245,E2 470.4461} C_DIS
LIN {X 128.5156,Y -52.9851,Z 174,A -20.3368,B 7.7687,C 0.3152,E1 7.9227,E2 472.2059} C_DIS
LIN {X 125.1226,Y -60.5649,Z 174,A -23.7916,B 7.7683,C 0.325,E1 7.9187,E2 475.6683} C_DIS
LIN {X 122.742,Y -65.2545,Z 174,A -25.9565,B 7.768,C 0.3305,E1 7.916,E2 477.835} C_DIS
LIN {X 120.6176,Y -69.1035,Z 174,A -27.756,B 7.7678,C 0.3349,E1 7.9135,E2 479.6347} C_DIS
LIN {X 119.1129,Y -71.6662,Z 174,A -29.1916,B 7.7675,C 0.3423,E1 7.9114,E2 481.0987} C_DIS
LIN {X 117.3489,Y -74.5198,Z 174,A -30.3691,B 7.7675,C 0.3416,E1 7.9097,E2 482.2512} C_DIS
LIN {X 114.848,Y -78.3194,Z 174,A -32.2257,B 7.7674,C 0.3458,E1 7.9068,E2 484.1073} C_DIS
LIN {X 112.5116,Y -81.6392,Z 174,A -33.7239,B 7.7674,C 0.3463,E1 7.9044,E2 485.5846} C_DIS
LIN {X 110.4994,Y -84.3424,Z 174,A -35.581,B 7.7668,C 0.3589,E1 7.9011,E2 487.5033} C_DIS
LIN {X 107.8296,Y -87.7308,Z 174,A -36.9495,B 7.767,C 0.3549,E1 7.8988,E2 488.8208} C_DIS
LIN {X 103.7915,Y -92.4731,Z 174,A -39.4578,B 7.7667,C 0.3595,E1 7.8943,E2 491.3241} C_DIS
LIN {X 98.9733,Y -97.6127,Z 174,A -42.3773,B 7.7664,C 0.3661,E1 7.8886,E2 494.2485} C_DIS
LIN {X 95.6964,Y -100.8276,Z 174,A -44.206,B 7.7664,C 0.3688,E1 7.885,E2 496.0708} C_DIS
LIN {X 92.5127,Y -103.7558,Z 174,A -46.5222,B 7.7656,C 0.3828,E1 7.88,E2 498.4573} C_DIS
LIN {X 88.5626,Y -107.1471,Z 174,A -48.0956,B 7.766,C 0.3758,E1 7.8768,E2 499.959} C_DIS
LIN {X 85.7566,Y -109.4059,Z 174,A -49.885,B 7.7656,C 0.3845,E1 7.8728,E2 501.7891} C_DIS
LIN {X 82.5749,Y -111.8272,Z 174,A -51.82,B 7.7651,C 0.393,E1 7.8683,E2 503.7625} C_DIS
LIN {X 77.9617,Y -115.0904,Z 174,A -53.4924,B 7.7656,C 0.3844,E1 7.8647,E2 505.3523} C_DIS
LIN {X 74.7168,Y -117.2233,Z 174,A -55.8596,B 7.7647,C 0.4017,E1 7.8589,E2 507.8196} C_DIS
LIN {X 69.1395,Y -120.5971,Z 174,A -57.7716,B 7.7652,C 0.3911,E1 7.8545,E2 509.6344} C_DIS
LIN {X 65.1615,Y -122.7909,Z 174,A -59.6015,B 7.7652,C 0.393,E1 7.85,E2 511.4603} C_DIS
LIN {X 62.3713,Y -124.2324,Z 174,A -60.8888,B 7.765,C 0.3947,E1 7.8468,E2 512.7478} C_DIS
LIN {X 58.6967,Y -126.0084,Z 174,A -62.2877,B 7.7652,C 0.3916,E1 7.8434,E2 514.1112} C_DIS
LIN {X 56.0941,Y -127.1884,Z 174,A -63.8896,B 7.7647,C 0.4011,E1 7.8391,E2 515.769} C_DIS
LIN {X 51.0895,Y -129.2817,Z 174,A -65.8383,B 7.7649,C 0.3984,E1 7.8342,E2 517.6823} C_DIS
LIN {X 47.6063,Y -130.6031,Z 174,A -67.5986,B 7.7646,C 0.4043,E1 7.8295,E2 519.4729} C_DIS
LIN {X 41.4928,Y -132.6739,Z 174,A -70.1441,B 7.7646,C 0.4049,E1 7.8228,E2 522.0054} C_DIS
LIN {X 37.5962,Y -133.8278,Z 174,A -71.6629,B 7.7646,C 0.4035,E1 7.8187,E2 523.505} C_DIS
LIN {X 30.0126,Y -135.7316,Z 174,A -74.9847,B 7.7644,C 0.4079,E1 7.8097,E2 526.842} C_DIS
LIN {X 23.3044,Y -137.0418,Z 174,A -78.1171,B 7.764,C 0.4154,E1 7.801,E2 530.0168} C_DIS
LIN {X 19.2816,Y -137.6653,Z 174,A -79.4701,B 7.7642,C 0.4105,E1 7.7973,E2 531.3288} C_DIS
LIN {X 15.4391,Y -138.1497,Z 174,A -81.0111,B 7.7642,C 0.4102,E1 7.7931,E2 532.8636} C_DIS
LIN {X 11.69,Y -138.5162,Z 174,A -82.5341,B 7.7642,C 0.4102,E1 7.7889,E2 534.3835} C_DIS
LIN {X 7.4107,Y -138.8117,Z 174,A -84.2823,B 7.7642,C 0.4105,E1 7.784,E2 536.1301} C_DIS
LIN {X 3.8443,Y -138.9555,Z 174,A -85.7497,B 7.7642,C 0.4107,E1 7.7799,E2 537.5978} C_DIS
LIN {X 0.9845,Y -139.0008,Z 174,A -86.6636,B 7.7645,C 0.4062,E1 7.7774,E2 538.4776} C_DIS
Enddeposition()
LIN {X 0.9845,Y -139.0008,Z 174,A -86.6636,B 7.7645,C 0.4062,E1 7.7774,E2 538.4776} C_DIS
Startdeposition()
$VEL.CP = VEL_PRINT
LIN {X 2.4259,Y -139.8949,Z 174,A -85.6186,B 7.704,C 0.403,E1 7.7198,E2 537.4236} C_DIS
LIN {X 6.5896,Y -139.7612,Z 174,A -83.8967,B 7.704,C 0.4023,E1 7.7247,E2 535.6988} C_DIS
LIN {X 10.2286,Y -139.5414,Z 174,A -82.3969,B 7.704,C 0.4017,E1 7.7288,E2 534.1972} C_DIS
LIN {X 14.8337,Y -139.1272,Z 174,A -80.528,B 7.7041,C 0.4014,E1 7.734,E2 532.3305} C_DIS
LIN {X 17.7057,Y -138.7917,Z 174,A -78.8698,B 7.7046,C 0.3922,E1 7.7388,E2 530.6086} C_DIS
LIN {X 22.3009,Y -138.1289,Z 174,A -77.535,B 7.7041,C 0.4015,E1 7.7423,E2 529.3481} C_DIS
LIN {X 27.205,Y -137.2471,Z 174,A -75.36,B 7.7043,C 0.3977,E1 7.7483,E2 527.154} C_DIS
LIN {X 31.1032,Y -136.4146,Z 174,A -73.2175,B 7.7048,C 0.387,E1 7.7543,E2 524.9424} C_DIS
LIN {X 36.0991,Y -135.1784,Z 174,A -71.7008,B 7.7044,C 0.3963,E1 7.7582,E2 523.503} C_DIS
LIN {X 40.2362,Y -134.0072,Z 174,A -69.9169,B 7.7044,C 0.3942,E1 7.763,E2 521.7149} C_DIS
LIN {X 47.323,Y -131.6695,Z 174,A -66.9602,B 7.7045,C 0.3929,E1 7.7708,E2 518.7691} C_DIS
LIN {X 50.2406,Y -130.5849,Z 174,A -65.61,B 7.7047,C 0.3901,E1 7.7744,E2 517.408} C_DIS
LIN {X 54.3708,Y -128.92,Z 174,A -63.3386,B 7.7052,C 0.3793,E1 7.7804,E2 515.0756} C_DIS
LIN {X 58.6464,Y -127.0311,Z 174,A -62.017,B 7.7048,C 0.3882,E1 7.7835,E2 513.8313} C_DIS
LIN {X 61.5719,Y -125.6396,Z 174,A -60.5994,B 7.705,C 0.3846,E1 7.7871,E2 512.4006} C_DIS
LIN {X 64.7887,Y -124.0112,Z 174,A -59.2138,B 7.705,C 0.3843,E1 7.7905,E2 511.0259} C_DIS
LIN {X 68.5181,Y -121.9923,Z 174,A -57.3939,B 7.7052,C 0.3801,E1 7.795,E2 509.1935} C_DIS
LIN {X 75.233,Y -117.9699,Z 174,A -54.1179,B 7.7055,C 0.3736,E1 7.8029,E2 505.9055} C_DIS
LIN {X 78.7913,Y -115.6234,Z 174,A -52.2254,B 7.7058,C 0.3677,E1 7.8073,E2 503.9919} C_DIS
LIN {X 81.836,Y -113.4888,Z 174,A -50.8643,B 7.7058,C 0.3682,E1 7.8103,E2 502.6509} C_DIS
LIN {X 86.0424,Y -110.3346,Z 174,A -48.858,B 7.7058,C 0.3671,E1 7.8147,E2 500.6622} C_DIS
LIN {X 89.4322,Y -107.6047,Z 174,A -47.3626,B 7.7057,C 0.3694,E1 7.8179,E2 499.203} C_DIS
LIN {X 92.4856,Y -104.9919,Z 174,A -45.3279,B 7.7062,C 0.3585,E1 7.8223,E2 497.1154} C_DIS
LIN {X 96.2751,Y -101.5287,Z 174,A -43.3651,B 7.7062,C 0.3569,E1 7.8263,E2 495.1691} C_DIS
LIN {X 99.6144,Y -98.2547,Z 174,A -41.727,B 7.7062,C 0.3584,E1 7.8294,E2 493.5658} C_DIS
LIN {X 102.4867,Y -95.2541,Z 174,A -39.5324,B 7.7068,C 0.3448,E1 7.8338,E2 491.3042} C_DIS
LIN {X 105.1439,Y -92.3135,Z 174,A -38.2088,B 7.7068,C 0.3473,E1 7.8362,E2 490.0187} C_DIS
LIN {X 108.1153,Y -88.8147,Z 174,A -36.4991,B 7.7068,C 0.3464,E1 7.8392,E2 488.3296} C_DIS
LIN {X 112.0876,Y -83.7448,Z 174,A -33.9396,B 7.707,C 0.3418,E1 7.8435,E2 485.7779} C_DIS
LIN {X 114.5464,Y -80.3498,Z 174,A -32.0424,B 7.7073,C 0.334,E1 7.8467,E2 483.8552} C_DIS
LIN {X 117.1761,Y -76.4638,Z 174,A -30.1528,B 7.7075,C 0.33,E1 7.8496,E2 481.968} C_DIS
LIN {X 119.948,Y -72.0383,Z 174,A -28.0894,B 7.7076,C 0.3261,E1 7.8526,E2 479.9123} C_DIS
Enddeposition()
END
